LIN {X 0,Y 720.163,Z 331.517,A -85,B 0,C 180,E1 -1485.703,E2 -1485.703} C_VEL
LIN {X 0,Y 720.147,Z 331.521,A -85,B 0,C 180,E1 -1488.211,E2 -1488.211} C_VEL
LIN {X 0,Y 720.224,Z 331.521,A -85,B 0,C 180,E1 -1491.031,E2 -1491.031} C_VEL
LIN {X 0,Y 720.178,Z 331.657,A -85,B 0,C 180,E1 -1491.842,E2 -1491.842} C_VEL
LIN {X 0,Y 724.726,Z 343.937,A -85,B 0,C 180,E1 -1493.02,E2 -1493.02} C_VEL
LIN {X 0,Y 724.3,Z 377.381,A -85,B 0,C 180,E1 -1495.364,E2 -1495.364} C_VEL
LIN {X 0,Y 726.478,Z 386.978,A -85,B 0,C 180,E1 -1495.595,E2 -1495.595} C_VEL
LIN {X 0,Y 725.424,Z 646.257,A -85,B 0,C 180,E1 -1498.535,E2 -1498.535} C_VEL
LIN {X 0,Y 724.936,Z 767.062,A -85,B 0,C 180,E1 -1499.901,E2 -1499.901} C_VEL
LIN {X 0,Y 724.615,Z 792.765,A -85,B 0,C 180,E1 -1500.336,E2 -1500.336} C_VEL
LIN {X 0,Y 724.343,Z 814.335,A -85,B 0,C 180,E1 -1500.838,E2 -1500.838} C_VEL
LIN {X 0,Y 723.978,Z 838.569,A -85,B 0,C 180,E1 -1501.544,E2 -1501.544} C_VEL
LIN {X 0,Y 723.547,Z 860.48,A -85,B 0,C 180,E1 -1502.333,E2 -1502.333} C_VEL
LIN {X 0,Y 723.146,Z 883.178,A -85,B 0,C 180,E1 -1503.296,E2 -1503.296} C_VEL
LIN {X 0,Y 722.632,Z 904.751,A -85,B 0,C 180,E1 -1504.38,E2 -1504.38} C_VEL
LIN {X 0,Y 722.216,Z 925.848,A -85,B 0,C 180,E1 -1505.596,E2 -1505.596} C_VEL
LIN {X 0,Y 721.746,Z 945.563,A -85,B 0,C 180,E1 -1506.911,E2 -1506.911} C_VEL
LIN {X 0,Y 721.365,Z 964.777,A -85,B 0,C 180,E1 -1508.364,E2 -1508.364} C_VEL
LIN {X 0,Y 721.013,Z 981.39,A -85,B 0,C 180,E1 -1509.799,E2 -1509.799} C_VEL
LIN {X 0,Y 720.713,Z 998.517,A -85,B 0,C 180,E1 -1511.476,E2 -1511.476} C_VEL
LIN {X 0,Y 720.475,Z 1012.01,A -85,B 0,C 180,E1 -1512.982,E2 -1512.982} C_VEL
LIN {X 0,Y 720.287,Z 1026.218,A -85,B 0,C 180,E1 -1514.789,E2 -1514.789} C_VEL
LIN {X 0,Y 720.15,Z 1037.315,A -85,B 0,C 180,E1 -1516.429,E2 -1516.429} C_VEL
LIN {X 0,Y 720.044,Z 1047.962,A -85,B 0,C 180,E1 -1518.238,E2 -1518.238} C_VEL
LIN {X 0,Y 719.961,Z 1056.892,A -85,B 0,C 180,E1 -1520.083,E2 -1520.083} C_VEL
LIN {X 0,Y 719.941,Z 1063.423,A -85,B 0,C 180,E1 -1521.695,E2 -1521.695} C_VEL
LIN {X 0,Y 719.913,Z 1069.864,A -85,B 0,C 180,E1 -1523.701,E2 -1523.701} C_VEL
LIN {X 0,Y 719.916,Z 1073.813,A -85,B 0,C 180,E1 -1525.379,E2 -1525.379} C_VEL
LIN {X 0,Y 719.907,Z 1076.797,A -85,B 0,C 180,E1 -1527.214,E2 -1527.214} C_VEL
LIN {X 0,Y 719.9,Z 1078.284,A -85,B 0,C 180,E1 -1529.204,E2 -1529.204} C_VEL
LIN {X 0,Y 719.906,Z 1078.262,A -85,B 0,C 180,E1 -1530.875,E2 -1530.875} C_VEL
LIN {X 0,Y 719.913,Z 1076.572,A -85,B 0,C 180,E1 -1532.946,E2 -1532.946} C_VEL
LIN {X 0,Y 719.919,Z 1073.654,A -85,B 0,C 180,E1 -1534.7,E2 -1534.7} C_VEL
LIN {X 0,Y 719.908,Z 1069.015,A -85,B 0,C 180,E1 -1536.62,E2 -1536.62} C_VEL
LIN {X 0,Y 719.933,Z 1062.815,A -85,B 0,C 180,E1 -1538.466,E2 -1538.466} C_VEL
LIN {X 0,Y 719.974,Z 1056.182,A -85,B 0,C 180,E1 -1540.078,E2 -1540.078} C_VEL
LIN {X 0,Y 720.049,Z 1046.492,A -85,B 0,C 180,E1 -1542.022,E2 -1542.022} C_VEL
LIN {X 0,Y 720.154,Z 1036.797,A -85,B 0,C 180,E1 -1543.653,E2 -1543.653} C_VEL
LIN {X 0,Y 720.323,Z 1024.443,A -85,B 0,C 180,E1 -1545.457,E2 -1545.457} C_VEL
LIN {X 0,Y 720.483,Z 1011.221,A -85,B 0,C 180,E1 -1547.11,E2 -1547.11} C_VEL
LIN {X 0,Y 720.769,Z 996.177,A -85,B 0,C 180,E1 -1548.774,E2 -1548.774} C_VEL
LIN {X 0,Y 721.055,Z 979.534,A -85,B 0,C 180,E1 -1550.369,E2 -1550.369} C_VEL
LIN {X 0,Y 721.431,Z 961.606,A -85,B 0,C 180,E1 -1551.89,E2 -1551.89} C_VEL
LIN {X 0,Y 721.806,Z 943.238,A -85,B 0,C 180,E1 -1553.253,E2 -1553.253} C_VEL
LIN {X 0,Y 722.274,Z 921.437,A -85,B 0,C 180,E1 -1554.67,E2 -1554.67} C_VEL
LIN {X 0,Y 722.724,Z 901.529,A -85,B 0,C 180,E1 -1555.792,E2 -1555.792} C_VEL
LIN {X 0,Y 723.206,Z 878.258,A -85,B 0,C 180,E1 -1556.923,E2 -1556.923} C_VEL
LIN {X 0,Y 723.622,Z 857.112,A -85,B 0,C 180,E1 -1557.798,E2 -1557.798} C_VEL
LIN {X 0,Y 724.075,Z 832.967,A -85,B 0,C 180,E1 -1558.632,E2 -1558.632} C_VEL
LIN {X 0,Y 724.365,Z 811.106,A -85,B 0,C 180,E1 -1559.246,E2 -1559.246} C_VEL
LIN {X 0,Y 724.75,Z 786.453,A -85,B 0,C 180,E1 -1559.787,E2 -1559.787} C_VEL
LIN {X 0,Y 724.95,Z 763.825,A -85,B 0,C 180,E1 -1560.142,E2 -1560.142} C_VEL
LIN {X 0,Y 725.946,Z 508.893,A -85,B 0,C 180,E1 -1563.013,E2 -1563.013} C_VEL
LIN {X 0,Y 726.28,Z 385.255,A -85,B 0,C 180,E1 -1564.436,E2 -1564.436} C_VEL
LIN {X 0,Y 724.228,Z 376.686,A -85,B 0,C 180,E1 -1564.668,E2 -1564.668} C_VEL
LIN {X 0,Y 724.705,Z 343.754,A -85,B 0,C 180,E1 -1566.995,E2 -1566.995} C_VEL
LIN {X 0,Y 720.161,Z 331.519,A -85,B 0,C 180,E1 -1568.182,E2 -1568.182} C_VEL
LIN {X 0,Y 720.198,Z 331.523,A -85,B 0,C 180,E1 -1571.193,E2 -1571.193} C_VEL
LIN {X 0,Y 720.148,Z 331.519,A -85,B 0,C 180,E1 -1573.895,E2 -1573.895} C_VEL
LIN {X 0,Y 720.193,Z 331.516,A -85,B 0,C 180,E1 -1576.588,E2 -1576.588} C_VEL
LIN {X 0,Y 720.169,Z 331.519,A -85,B 0,C 180,E1 -1579.58,E2 -1579.58} C_VEL
LIN {X 0,Y 720.148,Z 331.518,A -85,B 0,C 180,E1 -1582.143,E2 -1582.143} C_VEL
LIN {X 0,Y 720.215,Z 331.502,A -85,B 0,C 180,E1 -1584.917,E2 -1584.917} C_VEL
LIN {X 0,Y 720.156,Z 331.518,A -85,B 0,C 180,E1 -1587.881,E2 -1587.881} C_VEL
LIN {X 0,Y 720.152,Z 331.517,A -85,B 0,C 180,E1 -1590.377,E2 -1590.377} C_VEL
LIN {X 0,Y 720.225,Z 331.513,A -85,B 0,C 180,E1 -1593.212,E2 -1593.212} C_VEL
LIN {X 0,Y 720.155,Z 331.517,A -85,B 0,C 180,E1 -1596.082,E2 -1596.082} C_VEL
LIN {X 0,Y 720.162,Z 331.516,A -85,B 0,C 180,E1 -1598.668,E2 -1598.668} C_VEL
LIN {X 0,Y 720.211,Z 331.523,A -85,B 0,C 180,E1 -1601.63,E2 -1601.63} C_VEL
LIN {X 0,Y 720.149,Z 331.517,A -85,B 0,C 180,E1 -1604.374,E2 -1604.374} C_VEL
LIN {X 0,Y 720.181,Z 331.515,A -85,B 0,C 180,E1 -1607.002,E2 -1607.002} C_VEL
LIN {X 0,Y 720.172,Z 331.521,A -85,B 0,C 180,E1 -1610.086,E2 -1610.086} C_VEL
LIN {X 0,Y 720.151,Z 331.513,A -85,B 0,C 180,E1 -1612.661,E2 -1612.661} C_VEL
LIN {X 0,Y 720.219,Z 331.515,A -85,B 0,C 180,E1 -1615.461,E2 -1615.461} C_VEL
LIN {X 0,Y 720.159,Z 331.519,A -85,B 0,C 180,E1 -1618.409,E2 -1618.409} C_VEL
LIN {X 0,Y 720.157,Z 331.516,A -85,B 0,C 180,E1 -1620.955,E2 -1620.955} C_VEL
LIN {X 0,Y 720.222,Z 331.517,A -85,B 0,C 180,E1 -1623.821,E2 -1623.821} C_VEL
LIN {X 0,Y 720.156,Z 331.515,A -85,B 0,C 180,E1 -1626.618,E2 -1626.618} C_VEL
LIN {X 0,Y 720.164,Z 331.516,A -85,B 0,C 180,E1 -1629.19,E2 -1629.19} C_VEL
LIN {X 0,Y 720.209,Z 331.521,A -85,B 0,C 180,E1 -1632.208,E2 -1632.208} C_VEL
LIN {X 0,Y 720.153,Z 331.516,A -85,B 0,C 180,E1 -1634.966,E2 -1634.966} C_VEL
LIN {X 0,Y 720.21,Z 331.52,A -85,B 0,C 180,E1 -1636.267,E2 -1636.267} C_VEL
LIN {X 0,Y 719.173,Z 331.652,A -85,B 0,C 180,E1 -1636.88,E2 -1636.88} C_VEL
LIN {X 0,Y 712.742,Z 332.446,A -85,B 0,C 180,E1 -1638.597,E2 -1638.597} C_VEL
LIN {X 0,Y 712.215,Z 332.505,A -85,B 0,C 180,E1 -1639.043,E2 -1639.043} C_VEL
LIN {X 0,Y 712.276,Z 332.502,A -85,B 0,C 180,E1 -1641.84,E2 -1641.84} C_VEL
LIN {X 0,Y 712.226,Z 332.509,A -85,B 0,C 180,E1 -1644.82,E2 -1644.82} C_VEL
LIN {X 0,Y 712.226,Z 332.503,A -85,B 0,C 180,E1 -1647.469,E2 -1647.469} C_VEL
LIN {X 0,Y 712.279,Z 332.508,A -85,B 0,C 180,E1 -1650.467,E2 -1650.467} C_VEL
LIN {X 0,Y 712.217,Z 332.507,A -85,B 0,C 180,E1 -1653.294,E2 -1653.294} C_VEL
LIN {X 0,Y 712.28,Z 332.503,A -85,B 0,C 180,E1 -1656.128,E2 -1656.128} C_VEL
LIN {X 0,Y 712.227,Z 332.509,A -85,B 0,C 180,E1 -1659.076,E2 -1659.076} C_VEL
LIN {X 0,Y 712.227,Z 332.506,A -85,B 0,C 180,E1 -1661.717,E2 -1661.717} C_VEL
LIN {X 0,Y 712.274,Z 332.509,A -85,B 0,C 180,E1 -1664.739,E2 -1664.739} C_VEL
LIN {X 0,Y 712.218,Z 332.509,A -85,B 0,C 180,E1 -1667.524,E2 -1667.524} C_VEL
LIN {X 0,Y 712.278,Z 332.506,A -85,B 0,C 180,E1 -1670.303,E2 -1670.303} C_VEL
LIN {X 0,Y 712.232,Z 332.508,A -85,B 0,C 180,E1 -1673.285,E2 -1673.285} C_VEL
LIN {X 0,Y 712.237,Z 332.645,A -85,B 0,C 180,E1 -1673.57,E2 -1673.57} C_VEL
LIN {X 0,Y 716.875,Z 346.54,A -85,B 0,C 180,E1 -1674.925,E2 -1674.925} C_VEL
LIN {X 0,Y 717.007,Z 348.113,A -85,B 0,C 180,E1 -1675.014,E2 -1675.014} C_VEL
LIN {X 0,Y 719.82,Z 359.371,A -85,B 0,C 180,E1 -1675.305,E2 -1675.305} C_VEL
LIN {X 0,Y 718.682,Z 598.601,A -85,B 0,C 180,E1 -1678.047,E2 -1678.047} C_VEL
LIN {X 0,Y 718.006,Z 736.954,A -85,B 0,C 180,E1 -1679.623,E2 -1679.623} C_VEL
LIN {X 0,Y 717.638,Z 762.534,A -85,B 0,C 180,E1 -1680.059,E2 -1680.059} C_VEL
LIN {X 0,Y 717.293,Z 784.195,A -85,B 0,C 180,E1 -1680.564,E2 -1680.564} C_VEL
LIN {X 0,Y 716.857,Z 808.586,A -85,B 0,C 180,E1 -1681.281,E2 -1681.281} C_VEL
LIN {X 0,Y 716.344,Z 830.47,A -85,B 0,C 180,E1 -1682.075,E2 -1682.075} C_VEL
LIN {X 0,Y 715.848,Z 853.086,A -85,B 0,C 180,E1 -1683.043,E2 -1683.043} C_VEL
LIN {X 0,Y 715.244,Z 874.745,A -85,B 0,C 180,E1 -1684.141,E2 -1684.141} C_VEL
LIN {X 0,Y 714.721,Z 895.739,A -85,B 0,C 180,E1 -1685.361,E2 -1685.361} C_VEL
LIN {X 0,Y 714.171,Z 915.623,A -85,B 0,C 180,E1 -1686.701,E2 -1686.701} C_VEL
LIN {X 0,Y 713.69,Z 934.764,A -85,B 0,C 180,E1 -1688.163,E2 -1688.163} C_VEL
LIN {X 0,Y 713.286,Z 950.904,A -85,B 0,C 180,E1 -1689.571,E2 -1689.571} C_VEL
LIN {X 0,Y 712.928,Z 967.586,A -85,B 0,C 180,E1 -1691.209,E2 -1691.209} C_VEL
LIN {X 0,Y 712.6,Z 982.184,A -85,B 0,C 180,E1 -1692.854,E2 -1692.854} C_VEL
LIN {X 0,Y 712.364,Z 996.488,A -85,B 0,C 180,E1 -1694.7,E2 -1694.7} C_VEL
LIN {X 0,Y 712.199,Z 1007.556,A -85,B 0,C 180,E1 -1696.358,E2 -1696.358} C_VEL
LIN {X 0,Y 712.08,Z 1018.068,A -85,B 0,C 180,E1 -1698.17,E2 -1698.17} C_VEL
LIN {X 0,Y 711.984,Z 1026.697,A -85,B 0,C 180,E1 -1699.971,E2 -1699.971} C_VEL
LIN {X 0,Y 711.943,Z 1033.255,A -85,B 0,C 180,E1 -1701.601,E2 -1701.601} C_VEL
LIN {X 0,Y 711.921,Z 1039.75,A -85,B 0,C 180,E1 -1703.63,E2 -1703.63} C_VEL
LIN {X 0,Y 711.915,Z 1043.884,A -85,B 0,C 180,E1 -1705.408,E2 -1705.408} C_VEL
LIN {X 0,Y 711.896,Z 1046.847,A -85,B 0,C 180,E1 -1707.263,E2 -1707.263} C_VEL
LIN {X 0,Y 711.901,Z 1048.272,A -85,B 0,C 180,E1 -1709.195,E2 -1709.195} C_VEL
LIN {X 0,Y 711.906,Z 1048.274,A -85,B 0,C 180,E1 -1710.885,E2 -1710.885} C_VEL
LIN {X 0,Y 711.905,Z 1046.747,A -85,B 0,C 180,E1 -1712.898,E2 -1712.898} C_VEL
LIN {X 0,Y 711.915,Z 1043.902,A -85,B 0,C 180,E1 -1714.673,E2 -1714.673} C_VEL
LIN {X 0,Y 711.914,Z 1039.772,A -85,B 0,C 180,E1 -1716.451,E2 -1716.451} C_VEL
LIN {X 0,Y 711.94,Z 1033.287,A -85,B 0,C 180,E1 -1718.48,E2 -1718.48} C_VEL
LIN {X 0,Y 711.991,Z 1026.718,A -85,B 0,C 180,E1 -1720.114,E2 -1720.114} C_VEL
LIN {X 0,Y 712.085,Z 1017.658,A -85,B 0,C 180,E1 -1721.995,E2 -1721.995} C_VEL
LIN {X 0,Y 712.204,Z 1007.079,A -85,B 0,C 180,E1 -1723.808,E2 -1723.808} C_VEL
LIN {X 0,Y 712.406,Z 994.78,A -85,B 0,C 180,E1 -1725.633,E2 -1725.633} C_VEL
LIN {X 0,Y 712.628,Z 980.892,A -85,B 0,C 180,E1 -1727.389,E2 -1727.389} C_VEL
LIN {X 0,Y 712.956,Z 965.781,A -85,B 0,C 180,E1 -1729.073,E2 -1729.073} C_VEL
LIN {X 0,Y 713.31,Z 950.02,A -85,B 0,C 180,E1 -1730.6,E2 -1730.6} C_VEL
LIN {X 0,Y 713.758,Z 932.179,A -85,B 0,C 180,E1 -1732.138,E2 -1732.138} C_VEL
LIN {X 0,Y 714.223,Z 913.86,A -85,B 0,C 180,E1 -1733.515,E2 -1733.515} C_VEL
LIN {X 0,Y 714.759,Z 893.636,A -85,B 0,C 180,E1 -1734.858,E2 -1734.858} C_VEL
LIN {X 0,Y 715.297,Z 873.155,A -85,B 0,C 180,E1 -1736.036,E2 -1736.036} C_VEL
LIN {X 0,Y 715.891,Z 850.245,A -85,B 0,C 180,E1 -1737.176,E2 -1737.176} C_VEL
LIN {X 0,Y 716.368,Z 829.357,A -85,B 0,C 180,E1 -1738.059,E2 -1738.059} C_VEL
LIN {X 0,Y 716.936,Z 805.882,A -85,B 0,C 180,E1 -1738.898,E2 -1738.898} C_VEL
LIN {X 0,Y 717.311,Z 782.472,A -85,B 0,C 180,E1 -1739.571,E2 -1739.571} C_VEL
LIN {X 0,Y 717.764,Z 758.503,A -85,B 0,C 180,E1 -1740.115,E2 -1740.115} C_VEL
LIN {X 0,Y 718.018,Z 734.505,A -85,B 0,C 180,E1 -1740.499,E2 -1740.499} C_VEL
LIN {X 0,Y 719.269,Z 474.983,A -85,B 0,C 180,E1 -1743.45,E2 -1743.45} C_VEL
LIN {X 0,Y 719.631,Z 357.815,A -85,B 0,C 180,E1 -1744.814,E2 -1744.814} C_VEL
LIN {X 0,Y 716.852,Z 347.387,A -85,B 0,C 180,E1 -1745.101,E2 -1745.101} C_VEL
LIN {X 0,Y 716.411,Z 344.69,A -85,B 0,C 180,E1 -1745.335,E2 -1745.335} C_VEL
LIN {X 0,Y 712.213,Z 332.514,A -85,B 0,C 180,E1 -1746.555,E2 -1746.555} C_VEL
LIN {X 0,Y 712.284,Z 332.507,A -85,B 0,C 180,E1 -1749.384,E2 -1749.384} C_VEL
LIN {X 0,Y 712.216,Z 332.509,A -85,B 0,C 180,E1 -1752.28,E2 -1752.28} C_VEL
LIN {X 0,Y 712.218,Z 332.502,A -85,B 0,C 180,E1 -1754.848,E2 -1754.848} C_VEL
LIN {X 0,Y 712.272,Z 332.494,A -85,B 0,C 180,E1 -1757.834,E2 -1757.834} C_VEL
LIN {X 0,Y 712.21,Z 332.507,A -85,B 0,C 180,E1 -1760.611,E2 -1760.611} C_VEL
LIN {X 0,Y 712.248,Z 332.508,A -85,B 0,C 180,E1 -1763.283,E2 -1763.283} C_VEL
LIN {X 0,Y 712.227,Z 332.505,A -85,B 0,C 180,E1 -1766.357,E2 -1766.357} C_VEL
LIN {X 0,Y 712.215,Z 332.506,A -85,B 0,C 180,E1 -1768.986,E2 -1768.986} C_VEL
LIN {X 0,Y 712.284,Z 332.503,A -85,B 0,C 180,E1 -1771.857,E2 -1771.857} C_VEL
LIN {X 0,Y 712.213,Z 332.507,A -85,B 0,C 180,E1 -1774.706,E2 -1774.706} C_VEL
LIN {X 0,Y 712.223,Z 332.507,A -85,B 0,C 180,E1 -1777.29,E2 -1777.29} C_VEL
LIN {X 0,Y 712.261,Z 332.501,A -85,B 0,C 180,E1 -1780.311,E2 -1780.311} C_VEL
LIN {X 0,Y 712.209,Z 332.507,A -85,B 0,C 180,E1 -1783.021,E2 -1783.021} C_VEL
LIN {X 0,Y 712.251,Z 332.507,A -85,B 0,C 180,E1 -1785.695,E2 -1785.695} C_VEL
LIN {X 0,Y 712.225,Z 332.501,A -85,B 0,C 180,E1 -1788.747,E2 -1788.747} C_VEL
LIN {X 0,Y 712.213,Z 332.508,A -85,B 0,C 180,E1 -1791.36,E2 -1791.36} C_VEL
LIN {X 0,Y 712.285,Z 332.506,A -85,B 0,C 180,E1 -1794.199,E2 -1794.199} C_VEL
LIN {X 0,Y 712.212,Z 332.506,A -85,B 0,C 180,E1 -1797.103,E2 -1797.103} C_VEL
LIN {X 0,Y 712.224,Z 332.506,A -85,B 0,C 180,E1 -1799.678,E2 -1799.678} C_VEL
LIN {X 0,Y 712.252,Z 332.499,A -85,B 0,C 180,E1 -1802.736,E2 -1802.736} C_VEL
LIN {X 0,Y 712.209,Z 332.508,A -85,B 0,C 180,E1 -1805.397,E2 -1805.397} C_VEL
LIN {X 0,Y 712.25,Z 332.507,A -85,B 0,C 180,E1 -1808.07,E2 -1808.07} C_VEL
LIN {X 0,Y 712.228,Z 332.504,A -85,B 0,C 180,E1 -1811.092,E2 -1811.092} C_VEL
LIN {X 0,Y 712.211,Z 332.507,A -85,B 0,C 180,E1 -1813.708,E2 -1813.708} C_VEL
LIN {X 0,Y 712.284,Z 332.504,A -85,B 0,C 180,E1 -1816.557,E2 -1816.557} C_VEL
LIN {X 0,Y 712.212,Z 332.506,A -85,B 0,C 180,E1 -1819.435,E2 -1819.435} C_VEL
LIN {X 0,Y 712.22,Z 332.507,A -85,B 0,C 180,E1 -1822.015,E2 -1822.015} C_VEL
LIN {X 0,Y 712.269,Z 332.503,A -85,B 0,C 180,E1 -1824.996,E2 -1824.996} C_VEL
LIN {X 0,Y 712.209,Z 332.505,A -85,B 0,C 180,E1 -1827.691,E2 -1827.691} C_VEL
LIN {X 0,Y 712.234,Z 332.511,A -85,B 0,C 180,E1 -1830.301,E2 -1830.301} C_VEL
LIN {X 0,Y 712.235,Z 332.505,A -85,B 0,C 180,E1 -1833.389,E2 -1833.389} C_VEL
LIN {X 0,Y 712.209,Z 332.509,A -85,B 0,C 180,E1 -1835.933,E2 -1835.933} C_VEL
LIN {X 0,Y 712.266,Z 332.512,A -85,B 0,C 180,E1 -1838.692,E2 -1838.692} C_VEL
LIN {X 0,Y 712.221,Z 332.504,A -85,B 0,C 180,E1 -1841.679,E2 -1841.679} C_VEL
LIN {X 0,Y 712.213,Z 332.508,A -85,B 0,C 180,E1 -1844.275,E2 -1844.275} C_VEL
LIN {X 0,Y 712.28,Z 332.506,A -85,B 0,C 180,E1 -1847.201,E2 -1847.201} C_VEL
LIN {X 0,Y 712.211,Z 332.512,A -85,B 0,C 180,E1 -1849.984,E2 -1849.984} C_VEL
LIN {X 0,Y 712.303,Z 332.751,A -85,B 0,C 180,E1 -1851.434,E2 -1851.434} C_VEL
LIN {X 0,Y 717.694,Z 347.21,A -85,B 0,C 180,E1 -1852.836,E2 -1852.836} C_VEL
LIN {X 0,Y 717.276,Z 377.476,A -85,B 0,C 180,E1 -1854.976,E2 -1854.976} C_VEL
LIN {X 0,Y 719.862,Z 388.764,A -85,B 0,C 180,E1 -1855.255,E2 -1855.255} C_VEL
LIN {X 0,Y 718.587,Z 648.03,A -85,B 0,C 180,E1 -1858.222,E2 -1858.222} C_VEL
LIN {X 0,Y 718.004,Z 767.169,A -85,B 0,C 180,E1 -1859.581,E2 -1859.581} C_VEL
LIN {X 0,Y 717.629,Z 792.892,A -85,B 0,C 180,E1 -1860.021,E2 -1860.021} C_VEL
LIN {X 0,Y 717.29,Z 814.457,A -85,B 0,C 180,E1 -1860.526,E2 -1860.526} C_VEL
LIN {X 0,Y 716.861,Z 838.566,A -85,B 0,C 180,E1 -1861.235,E2 -1861.235} C_VEL
LIN {X 0,Y 716.339,Z 860.484,A -85,B 0,C 180,E1 -1862.031,E2 -1862.031} C_VEL
LIN {X 0,Y 715.831,Z 883.581,A -85,B 0,C 180,E1 -1863.022,E2 -1863.022} C_VEL
LIN {X 0,Y 715.246,Z 904.755,A -85,B 0,C 180,E1 -1864.096,E2 -1864.096} C_VEL
LIN {X 0,Y 714.719,Z 925.754,A -85,B 0,C 180,E1 -1865.317,E2 -1865.317} C_VEL
LIN {X 0,Y 714.178,Z 945.151,A -85,B 0,C 180,E1 -1866.622,E2 -1866.622} C_VEL
LIN {X 0,Y 713.724,Z 963.808,A -85,B 0,C 180,E1 -1868.038,E2 -1868.038} C_VEL
LIN {X 0,Y 713.296,Z 980.461,A -85,B 0,C 180,E1 -1869.485,E2 -1869.485} C_VEL
LIN {X 0,Y 712.939,Z 996.965,A -85,B 0,C 180,E1 -1871.096,E2 -1871.096} C_VEL
LIN {X 0,Y 712.623,Z 1011.222,A -85,B 0,C 180,E1 -1872.695,E2 -1872.695} C_VEL
LIN {X 0,Y 712.408,Z 1025.06,A -85,B 0,C 180,E1 -1874.45,E2 -1874.45} C_VEL
LIN {X 0,Y 712.209,Z 1036.796,A -85,B 0,C 180,E1 -1876.192,E2 -1876.192} C_VEL
LIN {X 0,Y 712.082,Z 1046.948,A -85,B 0,C 180,E1 -1877.923,E2 -1877.923} C_VEL
LIN {X 0,Y 711.99,Z 1056.524,A -85,B 0,C 180,E1 -1879.886,E2 -1879.886} C_VEL
LIN {X 0,Y 711.94,Z 1063.119,A -85,B 0,C 180,E1 -1881.52,E2 -1881.52} C_VEL
LIN {X 0,Y 711.909,Z 1069.451,A -85,B 0,C 180,E1 -1883.467,E2 -1883.467} C_VEL
LIN {X 0,Y 711.918,Z 1073.813,A -85,B 0,C 180,E1 -1885.327,E2 -1885.327} C_VEL
LIN {X 0,Y 711.908,Z 1076.797,A -85,B 0,C 180,E1 -1887.182,E2 -1887.182} C_VEL
LIN {X 0,Y 711.901,Z 1078.284,A -85,B 0,C 180,E1 -1889.195,E2 -1889.195} C_VEL
LIN {X 0,Y 711.906,Z 1078.262,A -85,B 0,C 180,E1 -1890.885,E2 -1890.885} C_VEL
LIN {X 0,Y 711.913,Z 1076.572,A -85,B 0,C 180,E1 -1892.979,E2 -1892.979} C_VEL
LIN {X 0,Y 711.919,Z 1073.655,A -85,B 0,C 180,E1 -1894.753,E2 -1894.753} C_VEL
LIN {X 0,Y 711.913,Z 1069.015,A -85,B 0,C 180,E1 -1896.694,E2 -1896.694} C_VEL
LIN {X 0,Y 711.938,Z 1062.815,A -85,B 0,C 180,E1 -1898.562,E2 -1898.562} C_VEL
LIN {X 0,Y 712.001,Z 1056.183,A -85,B 0,C 180,E1 -1900.192,E2 -1900.192} C_VEL
LIN {X 0,Y 712.095,Z 1046.032,A -85,B 0,C 180,E1 -1902.241,E2 -1902.241} C_VEL
LIN {X 0,Y 712.214,Z 1036.279,A -85,B 0,C 180,E1 -1903.891,E2 -1903.891} C_VEL
LIN {X 0,Y 712.423,Z 1023.807,A -85,B 0,C 180,E1 -1905.716,E2 -1905.716} C_VEL
LIN {X 0,Y 712.64,Z 1010.515,A -85,B 0,C 180,E1 -1907.389,E2 -1907.389} C_VEL
LIN {X 0,Y 712.961,Z 995.334,A -85,B 0,C 180,E1 -1909.073,E2 -1909.073} C_VEL
LIN {X 0,Y 713.319,Z 979.534,A -85,B 0,C 180,E1 -1910.6,E2 -1910.6} C_VEL
LIN {X 0,Y 713.766,Z 961.607,A -85,B 0,C 180,E1 -1912.138,E2 -1912.138} C_VEL
LIN {X 0,Y 714.239,Z 943.238,A -85,B 0,C 180,E1 -1913.514,E2 -1913.514} C_VEL
LIN {X 0,Y 714.782,Z 922.167,A -85,B 0,C 180,E1 -1914.901,E2 -1914.901} C_VEL
LIN {X 0,Y 715.321,Z 902.335,A -85,B 0,C 180,E1 -1916.035,E2 -1916.035} C_VEL
LIN {X 0,Y 715.904,Z 879.256,A -85,B 0,C 180,E1 -1917.175,E2 -1917.175} C_VEL
LIN {X 0,Y 716.401,Z 858.24,A -85,B 0,C 180,E1 -1918.057,E2 -1918.057} C_VEL
LIN {X 0,Y 716.951,Z 834.44,A -85,B 0,C 180,E1 -1918.897,E2 -1918.897} C_VEL
LIN {X 0,Y 717.314,Z 811.862,A -85,B 0,C 180,E1 -1919.542,E2 -1919.542} C_VEL
LIN {X 0,Y 717.775,Z 787.54,A -85,B 0,C 180,E1 -1920.087,E2 -1920.087} C_VEL
LIN {X 0,Y 718.02,Z 764.119,A -85,B 0,C 180,E1 -1920.459,E2 -1920.459} C_VEL
LIN {X 0,Y 719.22,Z 511.246,A -85,B 0,C 180,E1 -1923.334,E2 -1923.334} C_VEL
LIN {X 0,Y 719.678,Z 387.122,A -85,B 0,C 180,E1 -1924.775,E2 -1924.775} C_VEL
LIN {X 0,Y 717.183,Z 376.686,A -85,B 0,C 180,E1 -1925.058,E2 -1925.058} C_VEL
LIN {X 0,Y 717.694,Z 347.21,A -85,B 0,C 180,E1 -1927.164,E2 -1927.164} C_VEL
LIN {X 0,Y 712.275,Z 332.499,A -85,B 0,C 180,E1 -1928.608,E2 -1928.608} C_VEL
LIN {X 0,Y 712.219,Z 332.511,A -85,B 0,C 180,E1 -1931.558,E2 -1931.558} C_VEL
LIN {X 0,Y 712.213,Z 332.508,A -85,B 0,C 180,E1 -1934.134,E2 -1934.134} C_VEL
LIN {X 0,Y 712.282,Z 332.509,A -85,B 0,C 180,E1 -1937.001,E2 -1937.001} C_VEL
LIN {X 0,Y 712.215,Z 332.507,A -85,B 0,C 180,E1 -1939.794,E2 -1939.794} C_VEL
LIN {X 0,Y 712.22,Z 332.506,A -85,B 0,C 180,E1 -1942.36,E2 -1942.36} C_VEL
LIN {X 0,Y 712.269,Z 332.499,A -85,B 0,C 180,E1 -1945.351,E2 -1945.351} C_VEL
LIN {X 0,Y 712.21,Z 332.506,A -85,B 0,C 180,E1 -1948.043,E2 -1948.043} C_VEL
LIN {X 0,Y 712.236,Z 332.504,A -85,B 0,C 180,E1 -1950.669,E2 -1950.669} C_VEL
LIN {X 0,Y 712.236,Z 332.51,A -85,B 0,C 180,E1 -1953.776,E2 -1953.776} C_VEL
LIN {X 0,Y 712.213,Z 332.504,A -85,B 0,C 180,E1 -1956.414,E2 -1956.414} C_VEL
LIN {X 0,Y 712.281,Z 332.504,A -85,B 0,C 180,E1 -1959.215,E2 -1959.215} C_VEL
LIN {X 0,Y 712.219,Z 332.508,A -85,B 0,C 180,E1 -1962.147,E2 -1962.147} C_VEL
LIN {X 0,Y 712.219,Z 332.504,A -85,B 0,C 180,E1 -1964.696,E2 -1964.696} C_VEL
LIN {X 0,Y 712.282,Z 332.507,A -85,B 0,C 180,E1 -1967.597,E2 -1967.597} C_VEL
LIN {X 0,Y 712.214,Z 332.508,A -85,B 0,C 180,E1 -1970.383,E2 -1970.383} C_VEL
LIN {X 0,Y 712.231,Z 332.499,A -85,B 0,C 180,E1 -1972.999,E2 -1972.999} C_VEL
LIN {X 0,Y 712.25,Z 332.507,A -85,B 0,C 180,E1 -1976.056,E2 -1976.056} C_VEL
LIN {X 0,Y 712.214,Z 332.506,A -85,B 0,C 180,E1 -1978.713,E2 -1978.713} C_VEL
LIN {X 0,Y 712.272,Z 332.502,A -85,B 0,C 180,E1 -1981.448,E2 -1981.448} C_VEL
LIN {X 0,Y 712.228,Z 332.509,A -85,B 0,C 180,E1 -1984.428,E2 -1984.428} C_VEL
LIN {X 0,Y 712.217,Z 332.501,A -85,B 0,C 180,E1 -1987.016,E2 -1987.016} C_VEL
LIN {X 0,Y 712.283,Z 332.506,A -85,B 0,C 180,E1 -1989.861,E2 -1989.861} C_VEL
LIN {X 0,Y 712.22,Z 332.508,A -85,B 0,C 180,E1 -1992.733,E2 -1992.733} C_VEL
LIN {X 0,Y 712.228,Z 332.503,A -85,B 0,C 180,E1 -1995.319,E2 -1995.319} C_VEL
LIN {X 0,Y 712.267,Z 332.51,A -85,B 0,C 180,E1 -1998.328,E2 -1998.328} C_VEL
LIN {X 0,Y 712.215,Z 332.505,A -85,B 0,C 180,E1 -1999.043,E2 -1999.043} C_VEL
LIN {X 0,Y 711.23,Z 332.631,A -85,B 0,C 180,E1 -1999.663,E2 -1999.663} C_VEL
LIN {X 0,Y 704.844,Z 333.426,A -85,B 0,C 180,E1 -2001.399,E2 -2001.399} C_VEL
LIN {X 0,Y 704.338,Z 333.491,A -85,B 0,C 180,E1 -2001.85,E2 -2001.85} C_VEL
LIN {X 0,Y 704.285,Z 333.497,A -85,B 0,C 180,E1 -2004.85,E2 -2004.85} C_VEL
LIN {X 0,Y 704.288,Z 333.492,A -85,B 0,C 180,E1 -2007.478,E2 -2007.478} C_VEL
LIN {X 0,Y 704.336,Z 333.496,A -85,B 0,C 180,E1 -2010.491,E2 -2010.491} C_VEL
LIN {X 0,Y 704.279,Z 333.496,A -85,B 0,C 180,E1 -2013.329,E2 -2013.329} C_VEL
LIN {X 0,Y 704.344,Z 333.493,A -85,B 0,C 180,E1 -2016.197,E2 -2016.197} C_VEL
LIN {X 0,Y 704.288,Z 333.498,A -85,B 0,C 180,E1 -2019.077,E2 -2019.077} C_VEL
LIN {X 0,Y 704.291,Z 333.495,A -85,B 0,C 180,E1 -2021.747,E2 -2021.747} C_VEL
LIN {X 0,Y 704.33,Z 333.497,A -85,B 0,C 180,E1 -2024.78,E2 -2024.78} C_VEL
LIN {X 0,Y 704.279,Z 333.499,A -85,B 0,C 180,E1 -2027.484,E2 -2027.484} C_VEL
LIN {X 0,Y 704.339,Z 333.495,A -85,B 0,C 180,E1 -2030.296,E2 -2030.296} C_VEL
LIN {X 0,Y 704.32,Z 333.634,A -85,B 0,C 180,E1 -2033.172,E2 -2033.172} C_VEL
LIN {X 0,Y 709.368,Z 347.884,A -85,B 0,C 180,E1 -2034.578,E2 -2034.578} C_VEL
LIN {X 0,Y 711.003,Z 352.12,A -85,B 0,C 180,E1 -2034.723,E2 -2034.723} C_VEL
LIN {X 0,Y 713.229,Z 361.085,A -85,B 0,C 180,E1 -2034.958,E2 -2034.958} C_VEL
LIN {X 0,Y 711.884,Z 600.56,A -85,B 0,C 180,E1 -2037.728,E2 -2037.728} C_VEL
LIN {X 0,Y 711.097,Z 737.105,A -85,B 0,C 180,E1 -2039.298,E2 -2039.298} C_VEL
LIN {X 0,Y 710.679,Z 762.714,A -85,B 0,C 180,E1 -2039.738,E2 -2039.738} C_VEL
LIN {X 0,Y 710.263,Z 784.404,A -85,B 0,C 180,E1 -2040.249,E2 -2040.249} C_VEL
LIN {X 0,Y 709.759,Z 808.599,A -85,B 0,C 180,E1 -2040.966,E2 -2040.966} C_VEL
LIN {X 0,Y 709.163,Z 830.517,A -85,B 0,C 180,E1 -2041.768,E2 -2041.768} C_VEL
LIN {X 0,Y 708.557,Z 853.296,A -85,B 0,C 180,E1 -2042.753,E2 -2042.753} C_VEL
LIN {X 0,Y 707.875,Z 874.758,A -85,B 0,C 180,E1 -2043.851,E2 -2043.851} C_VEL
LIN {X 0,Y 707.237,Z 895.744,A -85,B 0,C 180,E1 -2045.083,E2 -2045.083} C_VEL
LIN {X 0,Y 706.626,Z 915.042,A -85,B 0,C 180,E1 -2046.394,E2 -2046.394} C_VEL
LIN {X 0,Y 706.047,Z 934.257,A -85,B 0,C 180,E1 -2047.87,E2 -2047.87} C_VEL
LIN {X 0,Y 705.56,Z 950.911,A -85,B 0,C 180,E1 -2049.337,E2 -2049.337} C_VEL
LIN {X 0,Y 705.123,Z 967.338,A -85,B 0,C 180,E1 -2050.965,E2 -2050.965} C_VEL
LIN {X 0,Y 704.759,Z 981.558,A -85,B 0,C 180,E1 -2052.581,E2 -2052.581} C_VEL
LIN {X 0,Y 704.49,Z 995.336,A -85,B 0,C 180,E1 -2054.356,E2 -2054.356} C_VEL
LIN {X 0,Y 704.268,Z 1007.041,A -85,B 0,C 180,E1 -2056.117,E2 -2056.117} C_VEL
LIN {X 0,Y 704.117,Z 1017.618,A -85,B 0,C 180,E1 -2057.951,E2 -2057.951} C_VEL
LIN {X 0,Y 704.01,Z 1026.7,A -85,B 0,C 180,E1 -2059.857,E2 -2059.857} C_VEL
LIN {X 0,Y 703.948,Z 1033.257,A -85,B 0,C 180,E1 -2061.505,E2 -2061.505} C_VEL
LIN {X 0,Y 703.922,Z 1039.544,A -85,B 0,C 180,E1 -2063.475,E2 -2063.475} C_VEL
LIN {X 0,Y 703.909,Z 1043.726,A -85,B 0,C 180,E1 -2065.274,E2 -2065.274} C_VEL
LIN {X 0,Y 703.911,Z 1046.51,A -85,B 0,C 180,E1 -2066.987,E2 -2066.987} C_VEL
LIN {X 0,Y 703.907,Z 1048.25,A -85,B 0,C 180,E1 -2069.105,E2 -2069.105} C_VEL
LIN {X 0,Y 703.902,Z 1048.296,A -85,B 0,C 180,E1 -2070.814,E2 -2070.814} C_VEL
LIN {X 0,Y 703.898,Z 1046.972,A -85,B 0,C 180,E1 -2072.768,E2 -2072.768} C_VEL
LIN {X 0,Y 703.916,Z 1044.06,A -85,B 0,C 180,E1 -2074.644,E2 -2074.644} C_VEL
LIN {X 0,Y 703.918,Z 1040.184,A -85,B 0,C 180,E1 -2076.361,E2 -2076.361} C_VEL
LIN {X 0,Y 703.95,Z 1033.892,A -85,B 0,C 180,E1 -2078.413,E2 -2078.413} C_VEL
LIN {X 0,Y 704.006,Z 1027.087,A -85,B 0,C 180,E1 -2080.144,E2 -2080.144} C_VEL
LIN {X 0,Y 704.115,Z 1018.105,A -85,B 0,C 180,E1 -2082.049,E2 -2082.049} C_VEL
LIN {X 0,Y 704.259,Z 1007.596,A -85,B 0,C 180,E1 -2083.883,E2 -2083.883} C_VEL
LIN {X 0,Y 704.475,Z 995.95,A -85,B 0,C 180,E1 -2085.645,E2 -2085.645} C_VEL
LIN {X 0,Y 704.741,Z 982.305,A -85,B 0,C 180,E1 -2087.42,E2 -2087.42} C_VEL
LIN {X 0,Y 705.1,Z 968.15,A -85,B 0,C 180,E1 -2089.036,E2 -2089.036} C_VEL
LIN {X 0,Y 705.546,Z 951.316,A -85,B 0,C 180,E1 -2090.715,E2 -2090.715} C_VEL
LIN {X 0,Y 706.047,Z 934.282,A -85,B 0,C 180,E1 -2092.217,E2 -2092.217} C_VEL
LIN {X 0,Y 706.624,Z 915.062,A -85,B 0,C 180,E1 -2093.695,E2 -2093.695} C_VEL
LIN {X 0,Y 707.258,Z 895.078,A -85,B 0,C 180,E1 -2095.051,E2 -2095.051} C_VEL
LIN {X 0,Y 707.906,Z 873.952,A -85,B 0,C 180,E1 -2096.283,E2 -2096.283} C_VEL
LIN {X 0,Y 708.585,Z 852.224,A -85,B 0,C 180,E1 -2097.389,E2 -2097.389} C_VEL
LIN {X 0,Y 709.16,Z 830.467,A -85,B 0,C 180,E1 -2098.324,E2 -2098.324} C_VEL
LIN {X 0,Y 709.784,Z 808.047,A -85,B 0,C 180,E1 -2099.142,E2 -2099.142} C_VEL
LIN {X 0,Y 710.27,Z 783.901,A -85,B 0,C 180,E1 -2099.855,E2 -2099.855} C_VEL
LIN {X 0,Y 710.715,Z 761.77,A -85,B 0,C 180,E1 -2100.371,E2 -2100.371} C_VEL
LIN {X 0,Y 711.1,Z 736.497,A -85,B 0,C 180,E1 -2100.8,E2 -2100.8} C_VEL
LIN {X 0,Y 712.564,Z 478.598,A -85,B 0,C 180,E1 -2103.764,E2 -2103.764} C_VEL
LIN {X 0,Y 713.042,Z 359.6,A -85,B 0,C 180,E1 -2105.161,E2 -2105.161} C_VEL
LIN {X 0,Y 709.992,Z 349.229,A -85,B 0,C 180,E1 -2105.46,E2 -2105.46} C_VEL
LIN {X 0,Y 709.099,Z 347.303,A -85,B 0,C 180,E1 -2105.548,E2 -2105.548} C_VEL
LIN {X 0,Y 704.3,Z 333.493,A -85,B 0,C 180,E1 -2106.937,E2 -2106.937} C_VEL
LIN {X 0,Y 704.296,Z 333.498,A -85,B 0,C 180,E1 -2110.025,E2 -2110.025} C_VEL
LIN {X 0,Y 704.274,Z 333.5,A -85,B 0,C 180,E1 -2112.656,E2 -2112.656} C_VEL
LIN {X 0,Y 704.345,Z 333.498,A -85,B 0,C 180,E1 -2115.566,E2 -2115.566} C_VEL
LIN {X 0,Y 704.273,Z 333.484,A -85,B 0,C 180,E1 -2118.469,E2 -2118.469} C_VEL
LIN {X 0,Y 704.298,Z 333.498,A -85,B 0,C 180,E1 -2121.133,E2 -2121.133} C_VEL
LIN {X 0,Y 704.301,Z 333.495,A -85,B 0,C 180,E1 -2124.203,E2 -2124.203} C_VEL
LIN {X 0,Y 704.273,Z 333.497,A -85,B 0,C 180,E1 -2126.893,E2 -2126.893} C_VEL
LIN {X 0,Y 704.347,Z 333.497,A -85,B 0,C 180,E1 -2129.738,E2 -2129.738} C_VEL
LIN {X 0,Y 704.278,Z 333.491,A -85,B 0,C 180,E1 -2132.613,E2 -2132.613} C_VEL
LIN {X 0,Y 704.277,Z 333.498,A -85,B 0,C 180,E1 -2135.15,E2 -2135.15} C_VEL
LIN {X 0,Y 704.343,Z 333.494,A -85,B 0,C 180,E1 -2138.077,E2 -2138.077} C_VEL
LIN {X 0,Y 704.274,Z 333.492,A -85,B 0,C 180,E1 -2140.855,E2 -2140.855} C_VEL
LIN {X 0,Y 704.295,Z 333.499,A -85,B 0,C 180,E1 -2143.504,E2 -2143.504} C_VEL
LIN {X 0,Y 704.295,Z 333.494,A -85,B 0,C 180,E1 -2146.62,E2 -2146.62} C_VEL
LIN {X 0,Y 704.272,Z 333.492,A -85,B 0,C 180,E1 -2149.281,E2 -2149.281} C_VEL
LIN {X 0,Y 704.344,Z 333.494,A -85,B 0,C 180,E1 -2152.167,E2 -2152.167} C_VEL
LIN {X 0,Y 704.275,Z 333.494,A -85,B 0,C 180,E1 -2155.032,E2 -2155.032} C_VEL
LIN {X 0,Y 704.284,Z 333.497,A -85,B 0,C 180,E1 -2157.64,E2 -2157.64} C_VEL
LIN {X 0,Y 704.321,Z 333.493,A -85,B 0,C 180,E1 -2160.651,E2 -2160.651} C_VEL
LIN {X 0,Y 704.269,Z 333.49,A -85,B 0,C 180,E1 -2163.337,E2 -2163.337} C_VEL
LIN {X 0,Y 704.313,Z 333.5,A -85,B 0,C 180,E1 -2166.03,E2 -2166.03} C_VEL
LIN {X 0,Y 704.288,Z 333.494,A -85,B 0,C 180,E1 -2169.067,E2 -2169.067} C_VEL
LIN {X 0,Y 704.272,Z 333.495,A -85,B 0,C 180,E1 -2171.631,E2 -2171.631} C_VEL
LIN {X 0,Y 704.346,Z 333.497,A -85,B 0,C 180,E1 -2174.495,E2 -2174.495} C_VEL
LIN {X 0,Y 704.277,Z 333.493,A -85,B 0,C 180,E1 -2177.346,E2 -2177.346} C_VEL
LIN {X 0,Y 704.278,Z 333.497,A -85,B 0,C 180,E1 -2179.922,E2 -2179.922} C_VEL
LIN {X 0,Y 704.341,Z 333.492,A -85,B 0,C 180,E1 -2182.891,E2 -2182.891} C_VEL
LIN {X 0,Y 704.271,Z 333.496,A -85,B 0,C 180,E1 -2185.66,E2 -2185.66} C_VEL
LIN {X 0,Y 704.301,Z 333.497,A -85,B 0,C 180,E1 -2188.332,E2 -2188.332} C_VEL
LIN {X 0,Y 704.286,Z 333.493,A -85,B 0,C 180,E1 -2191.433,E2 -2191.433} C_VEL
LIN {X 0,Y 704.271,Z 333.497,A -85,B 0,C 180,E1 -2194.013,E2 -2194.013} C_VEL
LIN {X 0,Y 704.345,Z 333.495,A -85,B 0,C 180,E1 -2196.905,E2 -2196.905} C_VEL
LIN {X 0,Y 704.272,Z 333.492,A -85,B 0,C 180,E1 -2199.818,E2 -2199.818} C_VEL
LIN {X 0,Y 704.285,Z 333.496,A -85,B 0,C 180,E1 -2202.417,E2 -2202.417} C_VEL
LIN {X 0,Y 704.312,Z 333.494,A -85,B 0,C 180,E1 -2205.467,E2 -2205.467} C_VEL
LIN {X 0,Y 704.27,Z 333.499,A -85,B 0,C 180,E1 -2208.142,E2 -2208.142} C_VEL
LIN {X 0,Y 704.337,Z 333.499,A -85,B 0,C 180,E1 -2210.961,E2 -2210.961} C_VEL
LIN {X 0,Y 710.716,Z 350.759,A -85,B 0,C 180,E1 -2212.673,E2 -2212.673} C_VEL
LIN {X 0,Y 710.234,Z 377.393,A -85,B 0,C 180,E1 -2214.576,E2 -2214.576} C_VEL
LIN {X 0,Y 713.272,Z 390.545,A -85,B 0,C 180,E1 -2214.908,E2 -2214.908} C_VEL
LIN {X 0,Y 711.768,Z 650.523,A -85,B 0,C 180,E1 -2217.91,E2 -2217.91} C_VEL
LIN {X 0,Y 711.095,Z 767.212,A -85,B 0,C 180,E1 -2219.254,E2 -2219.254} C_VEL
LIN {X 0,Y 710.676,Z 792.89,A -85,B 0,C 180,E1 -2219.697,E2 -2219.697} C_VEL
LIN {X 0,Y 710.261,Z 814.557,A -85,B 0,C 180,E1 -2220.208,E2 -2220.208} C_VEL
LIN {X 0,Y 709.764,Z 838.562,A -85,B 0,C 180,E1 -2220.92,E2 -2220.92} C_VEL
LIN {X 0,Y 709.159,Z 860.488,A -85,B 0,C 180,E1 -2221.722,E2 -2221.722} C_VEL
LIN {X 0,Y 708.561,Z 883.169,A -85,B 0,C 180,E1 -2222.701,E2 -2222.701} C_VEL
LIN {X 0,Y 707.877,Z 904.758,A -85,B 0,C 180,E1 -2223.806,E2 -2223.806} C_VEL
LIN {X 0,Y 707.237,Z 925.751,A -85,B 0,C 180,E1 -2225.038,E2 -2225.038} C_VEL
LIN {X 0,Y 706.621,Z 945.051,A -85,B 0,C 180,E1 -2226.349,E2 -2226.349} C_VEL
LIN {X 0,Y 706.067,Z 963.762,A -85,B 0,C 180,E1 -2227.783,E2 -2227.783} C_VEL
LIN {X 0,Y 705.558,Z 980.804,A -85,B 0,C 180,E1 -2229.282,E2 -2229.282} C_VEL
LIN {X 0,Y 705.129,Z 996.966,A -85,B 0,C 180,E1 -2230.879,E2 -2230.879} C_VEL
LIN {X 0,Y 704.773,Z 1011.223,A -85,B 0,C 180,E1 -2232.496,E2 -2232.496} C_VEL
LIN {X 0,Y 704.503,Z 1025.06,A -85,B 0,C 180,E1 -2234.271,E2 -2234.271} C_VEL
LIN {X 0,Y 704.267,Z 1036.797,A -85,B 0,C 180,E1 -2236.033,E2 -2236.033} C_VEL
LIN {X 0,Y 704.122,Z 1046.947,A -85,B 0,C 180,E1 -2237.785,E2 -2237.785} C_VEL
LIN {X 0,Y 704.017,Z 1056.538,A -85,B 0,C 180,E1 -2239.774,E2 -2239.774} C_VEL
LIN {X 0,Y 703.947,Z 1063.12,A -85,B 0,C 180,E1 -2241.423,E2 -2241.423} C_VEL
LIN {X 0,Y 703.913,Z 1069.451,A -85,B 0,C 180,E1 -2243.393,E2 -2243.393} C_VEL
LIN {X 0,Y 703.919,Z 1073.814,A -85,B 0,C 180,E1 -2245.274,E2 -2245.274} C_VEL
LIN {X 0,Y 703.909,Z 1076.797,A -85,B 0,C 180,E1 -2247.15,E2 -2247.15} C_VEL
LIN {X 0,Y 703.902,Z 1078.284,A -85,B 0,C 180,E1 -2249.186,E2 -2249.186} C_VEL
LIN {X 0,Y 703.907,Z 1078.262,A -85,B 0,C 180,E1 -2250.895,E2 -2250.895} C_VEL
LIN {X 0,Y 703.916,Z 1076.573,A -85,B 0,C 180,E1 -2253.013,E2 -2253.013} C_VEL
LIN {X 0,Y 703.919,Z 1073.655,A -85,B 0,C 180,E1 -2254.807,E2 -2254.807} C_VEL
LIN {X 0,Y 703.922,Z 1069.015,A -85,B 0,C 180,E1 -2256.771,E2 -2256.771} C_VEL
LIN {X 0,Y 703.945,Z 1062.816,A -85,B 0,C 180,E1 -2258.659,E2 -2258.659} C_VEL
LIN {X 0,Y 704.025,Z 1056.183,A -85,B 0,C 180,E1 -2260.309,E2 -2260.309} C_VEL
LIN {X 0,Y 704.135,Z 1046.031,A -85,B 0,C 180,E1 -2262.382,E2 -2262.382} C_VEL
LIN {X 0,Y 704.274,Z 1036.281,A -85,B 0,C 180,E1 -2264.05,E2 -2264.05} C_VEL
LIN {X 0,Y 704.516,Z 1023.805,A -85,B 0,C 180,E1 -2265.897,E2 -2265.897} C_VEL
LIN {X 0,Y 704.794,Z 1010.517,A -85,B 0,C 180,E1 -2267.589,E2 -2267.589} C_VEL
LIN {X 0,Y 705.159,Z 995.333,A -85,B 0,C 180,E1 -2269.292,E2 -2269.292} C_VEL
LIN {X 0,Y 705.592,Z 979.535,A -85,B 0,C 180,E1 -2270.836,E2 -2270.836} C_VEL
LIN {X 0,Y 706.116,Z 961.608,A -85,B 0,C 180,E1 -2272.39,E2 -2272.39} C_VEL
LIN {X 0,Y 706.659,Z 944.007,A -85,B 0,C 180,E1 -2273.726,E2 -2273.726} C_VEL
LIN {X 0,Y 707.287,Z 923.623,A -85,B 0,C 180,E1 -2275.094,E2 -2275.094} C_VEL
LIN {X 0,Y 707.908,Z 903.834,A -85,B 0,C 180,E1 -2276.244,E2 -2276.244} C_VEL
LIN {X 0,Y 708.586,Z 882.241,A -85,B 0,C 180,E1 -2277.343,E2 -2277.343} C_VEL
LIN {X 0,Y 709.195,Z 859.367,A -85,B 0,C 180,E1 -2278.322,E2 -2278.322} C_VEL
LIN {X 0,Y 709.833,Z 836.517,A -85,B 0,C 180,E1 -2279.149,E2 -2279.149} C_VEL
LIN {X 0,Y 710.283,Z 812.684,A -85,B 0,C 180,E1 -2279.842,E2 -2279.842} C_VEL
LIN {X 0,Y 710.8,Z 788.99,A -85,B 0,C 180,E1 -2280.384,E2 -2280.384} C_VEL
LIN {X 0,Y 711.11,Z 764.773,A -85,B 0,C 180,E1 -2280.778,E2 -2280.778} C_VEL
LIN {X 0,Y 712.515,Z 513.855,A -85,B 0,C 180,E1 -2283.659,E2 -2283.659} C_VEL
LIN {X 0,Y 713.088,Z 388.851,A -85,B 0,C 180,E1 -2285.122,E2 -2285.122} C_VEL
LIN {X 0,Y 710.16,Z 376.686,A -85,B 0,C 180,E1 -2285.457,E2 -2285.457} C_VEL
LIN {X 0,Y 710.659,Z 350.511,A -85,B 0,C 180,E1 -2287.349,E2 -2287.349} C_VEL
LIN {X 0,Y 704.336,Z 333.49,A -85,B 0,C 180,E1 -2289.038,E2 -2289.038} C_VEL
LIN {X 0,Y 704.271,Z 333.499,A -85,B 0,C 180,E1 -2291.858,E2 -2291.858} C_VEL
LIN {X 0,Y 704.313,Z 333.495,A -85,B 0,C 180,E1 -2294.547,E2 -2294.547} C_VEL
LIN {X 0,Y 704.287,Z 333.498,A -85,B 0,C 180,E1 -2297.595,E2 -2297.595} C_VEL
LIN {X 0,Y 704.273,Z 333.494,A -85,B 0,C 180,E1 -2300.185,E2 -2300.185} C_VEL
LIN {X 0,Y 704.345,Z 333.489,A -85,B 0,C 180,E1 -2303.057,E2 -2303.057} C_VEL
LIN {X 0,Y 704.277,Z 333.495,A -85,B 0,C 180,E1 -2305.889,E2 -2305.889} C_VEL
LIN {X 0,Y 704.283,Z 333.492,A -85,B 0,C 180,E1 -2308.502,E2 -2308.502} C_VEL
LIN {X 0,Y 704.326,Z 333.495,A -85,B 0,C 180,E1 -2311.51,E2 -2311.51} C_VEL
LIN {X 0,Y 704.272,Z 333.496,A -85,B 0,C 180,E1 -2314.25,E2 -2314.25} C_VEL
LIN {X 0,Y 704.328,Z 333.49,A -85,B 0,C 180,E1 -2317.02,E2 -2317.02} C_VEL
LIN {X 0,Y 704.284,Z 333.496,A -85,B 0,C 180,E1 -2320.027,E2 -2320.027} C_VEL
LIN {X 0,Y 704.28,Z 333.494,A -85,B 0,C 180,E1 -2322.654,E2 -2322.654} C_VEL
LIN {X 0,Y 704.344,Z 333.497,A -85,B 0,C 180,E1 -2325.615,E2 -2325.615} C_VEL
LIN {X 0,Y 704.274,Z 333.493,A -85,B 0,C 180,E1 -2328.452,E2 -2328.452} C_VEL
LIN {X 0,Y 704.317,Z 333.493,A -85,B 0,C 180,E1 -2331.18,E2 -2331.18} C_VEL
LIN {X 0,Y 704.29,Z 333.499,A -85,B 0,C 180,E1 -2334.215,E2 -2334.215} C_VEL
LIN {X 0,Y 704.277,Z 333.492,A -85,B 0,C 180,E1 -2336.826,E2 -2336.826} C_VEL
LIN {X 0,Y 704.346,Z 333.496,A -85,B 0,C 180,E1 -2339.756,E2 -2339.756} C_VEL
LIN {X 0,Y 704.276,Z 333.494,A -85,B 0,C 180,E1 -2342.604,E2 -2342.604} C_VEL
LIN {X 0,Y 704.303,Z 333.493,A -85,B 0,C 180,E1 -2345.295,E2 -2345.295} C_VEL
LIN {X 0,Y 704.297,Z 333.499,A -85,B 0,C 180,E1 -2348.409,E2 -2348.409} C_VEL
LIN {X 0,Y 704.277,Z 333.491,A -85,B 0,C 180,E1 -2351.05,E2 -2351.05} C_VEL
LIN {X 0,Y 704.345,Z 333.496,A -85,B 0,C 180,E1 -2353.965,E2 -2353.965} C_VEL
LIN {X 0,Y 704.279,Z 333.496,A -85,B 0,C 180,E1 -2356.836,E2 -2356.836} C_VEL
LIN {X 0,Y 704.299,Z 333.492,A -85,B 0,C 180,E1 -2359.494,E2 -2359.494} C_VEL
LIN {X 0,Y 704.338,Z 333.491,A -85,B 0,C 180,E1 -2361.85,E2 -2361.85} C_VEL
LIN {X 0,Y 703.383,Z 333.619,A -85,B 0,C 180,E1 -2362.476,E2 -2362.476} C_VEL
LIN {X 0,Y 696.932,Z 334.423,A -85,B 0,C 180,E1 -2364.231,E2 -2364.231} C_VEL
LIN {X 0,Y 696.359,Z 334.487,A -85,B 0,C 180,E1 -2364.688,E2 -2364.688} C_VEL
LIN {X 0,Y 696.343,Z 334.481,A -85,B 0,C 180,E1 -2367.355,E2 -2367.355} C_VEL
LIN {X 0,Y 696.407,Z 334.486,A -85,B 0,C 180,E1 -2370.263,E2 -2370.263} C_VEL
LIN {X 0,Y 696.341,Z 334.486,A -85,B 0,C 180,E1 -2373.168,E2 -2373.168} C_VEL
LIN {X 0,Y 696.384,Z 334.481,A -85,B 0,C 180,E1 -2375.963,E2 -2375.963} C_VEL
LIN {X 0,Y 696.353,Z 334.488,A -85,B 0,C 180,E1 -2379.03,E2 -2379.03} C_VEL
LIN {X 0,Y 696.349,Z 334.485,A -85,B 0,C 180,E1 -2381.697,E2 -2381.697} C_VEL
LIN {X 0,Y 696.398,Z 334.486,A -85,B 0,C 180,E1 -2384.712,E2 -2384.712} C_VEL
LIN {X 0,Y 696.341,Z 334.488,A -85,B 0,C 180,E1 -2387.555,E2 -2387.555} C_VEL
LIN {X 0,Y 696.404,Z 334.486,A -85,B 0,C 180,E1 -2390.395,E2 -2390.395} C_VEL
LIN {X 0,Y 696.428,Z 334.656,A -85,B 0,C 180,E1 -2392.751,E2 -2392.751} C_VEL
LIN {X 0,Y 701.14,Z 347.989,A -85,B 0,C 180,E1 -2394.098,E2 -2394.098} C_VEL
LIN {X 0,Y 704.659,Z 354.748,A -85,B 0,C 180,E1 -2394.389,E2 -2394.389} C_VEL
LIN {X 0,Y 706.664,Z 362.972,A -85,B 0,C 180,E1 -2394.606,E2 -2394.606} C_VEL
LIN {X 0,Y 705.107,Z 602.463,A -85,B 0,C 180,E1 -2397.401,E2 -2397.401} C_VEL
LIN {X 0,Y 704.211,Z 737.148,A -85,B 0,C 180,E1 -2398.965,E2 -2398.965} C_VEL
LIN {X 0,Y 703.748,Z 762.739,A -85,B 0,C 180,E1 -2399.409,E2 -2399.409} C_VEL
LIN {X 0,Y 703.256,Z 784.537,A -85,B 0,C 180,E1 -2399.925,E2 -2399.925} C_VEL
LIN {X 0,Y 702.684,Z 808.612,A -85,B 0,C 180,E1 -2400.646,E2 -2400.646} C_VEL
LIN {X 0,Y 702.042,Z 829.399,A -85,B 0,C 180,E1 -2401.409,E2 -2401.409} C_VEL
LIN {X 0,Y 701.346,Z 851.276,A -85,B 0,C 180,E1 -2402.351,E2 -2402.351} C_VEL
LIN {X 0,Y 700.587,Z 873.151,A -85,B 0,C 180,E1 -2403.467,E2 -2403.467} C_VEL
LIN {X 0,Y 699.872,Z 892.904,A -85,B 0,C 180,E1 -2404.621,E2 -2404.621} C_VEL
LIN {X 0,Y 699.15,Z 912.981,A -85,B 0,C 180,E1 -2405.973,E2 -2405.973} C_VEL
LIN {X 0,Y 698.518,Z 930.639,A -85,B 0,C 180,E1 -2407.32,E2 -2407.32} C_VEL
LIN {X 0,Y 697.901,Z 949.06,A -85,B 0,C 180,E1 -2408.924,E2 -2408.924} C_VEL
LIN {X 0,Y 697.39,Z 964.894,A -85,B 0,C 180,E1 -2410.484,E2 -2410.484} C_VEL
LIN {X 0,Y 696.961,Z 980.15,A -85,B 0,C 180,E1 -2412.207,E2 -2412.207} C_VEL
LIN {X 0,Y 696.62,Z 993.469,A -85,B 0,C 180,E1 -2413.918,E2 -2413.918} C_VEL
LIN {X 0,Y 696.353,Z 1006.007,A -85,B 0,C 180,E1 -2415.786,E2 -2415.786} C_VEL
LIN {X 0,Y 696.186,Z 1015.785,A -85,B 0,C 180,E1 -2417.475,E2 -2417.475} C_VEL
LIN {X 0,Y 696.048,Z 1025.993,A -85,B 0,C 180,E1 -2419.572,E2 -2419.572} C_VEL
LIN {X 0,Y 695.953,Z 1032.956,A -85,B 0,C 180,E1 -2421.324,E2 -2421.324} C_VEL
LIN {X 0,Y 695.936,Z 1039.125,A -85,B 0,C 180,E1 -2423.234,E2 -2423.234} C_VEL
LIN {X 0,Y 695.908,Z 1043.728,A -85,B 0,C 180,E1 -2425.22,E2 -2425.22} C_VEL
LIN {X 0,Y 695.912,Z 1046.511,A -85,B 0,C 180,E1 -2426.953,E2 -2426.953} C_VEL
LIN {X 0,Y 695.907,Z 1048.249,A -85,B 0,C 180,E1 -2429.094,E2 -2429.094} C_VEL
LIN {X 0,Y 695.902,Z 1048.296,A -85,B 0,C 180,E1 -2430.823,E2 -2430.823} C_VEL
LIN {X 0,Y 695.899,Z 1046.971,A -85,B 0,C 180,E1 -2432.8,E2 -2432.8} C_VEL
LIN {X 0,Y 695.916,Z 1044.059,A -85,B 0,C 180,E1 -2434.698,E2 -2434.698} C_VEL
LIN {X 0,Y 695.919,Z 1040.183,A -85,B 0,C 180,E1 -2436.435,E2 -2436.435} C_VEL
LIN {X 0,Y 695.954,Z 1033.89,A -85,B 0,C 180,E1 -2438.51,E2 -2438.51} C_VEL
LIN {X 0,Y 696.032,Z 1027.085,A -85,B 0,C 180,E1 -2440.261,E2 -2440.261} C_VEL
LIN {X 0,Y 696.153,Z 1018.102,A -85,B 0,C 180,E1 -2442.189,E2 -2442.189} C_VEL
LIN {X 0,Y 696.323,Z 1007.594,A -85,B 0,C 180,E1 -2444.045,E2 -2444.045} C_VEL
LIN {X 0,Y 696.572,Z 995.948,A -85,B 0,C 180,E1 -2445.827,E2 -2445.827} C_VEL
LIN {X 0,Y 696.894,Z 982.299,A -85,B 0,C 180,E1 -2447.622,E2 -2447.622} C_VEL
LIN {X 0,Y 697.295,Z 968.146,A -85,B 0,C 180,E1 -2449.257,E2 -2449.257} C_VEL
LIN {X 0,Y 697.808,Z 951.862,A -85,B 0,C 180,E1 -2450.903,E2 -2450.903} C_VEL
LIN {X 0,Y 698.361,Z 935.289,A -85,B 0,C 180,E1 -2452.386,E2 -2452.386} C_VEL
LIN {X 0,Y 699.032,Z 916.263,A -85,B 0,C 180,E1 -2453.879,E2 -2453.879} C_VEL
LIN {X 0,Y 699.697,Z 897.748,A -85,B 0,C 180,E1 -2455.159,E2 -2455.159} C_VEL
LIN {X 0,Y 700.465,Z 876.355,A -85,B 0,C 180,E1 -2456.447,E2 -2456.447} C_VEL
LIN {X 0,Y 701.167,Z 856.657,A -85,B 0,C 180,E1 -2457.477,E2 -2457.477} C_VEL
LIN {X 0,Y 701.929,Z 832.695,A -85,B 0,C 180,E1 -2458.549,E2 -2458.549} C_VEL
LIN {X 0,Y 702.549,Z 812.364,A -85,B 0,C 180,E1 -2459.314,E2 -2459.314} C_VEL
LIN {X 0,Y 703.221,Z 787.502,A -85,B 0,C 180,E1 -2460.086,E2 -2460.086} C_VEL
LIN {X 0,Y 703.676,Z 765.394,A -85,B 0,C 180,E1 -2460.625,E2 -2460.625} C_VEL
LIN {X 0,Y 704.188,Z 740.796,A -85,B 0,C 180,E1 -2461.076,E2 -2461.076} C_VEL
LIN {X 0,Y 704.537,Z 693.711,A -85,B 0,C 180,E1 -2461.643,E2 -2461.643} C_VEL
LIN {X 0,Y 706.175,Z 439.974,A -85,B 0,C 180,E1 -2464.576,E2 -2464.576} C_VEL
LIN {X 0,Y 706.502,Z 361.588,A -85,B 0,C 180,E1 -2465.51,E2 -2465.51} C_VEL
LIN {X 0,Y 703.94,Z 352.965,A -85,B 0,C 180,E1 -2465.765,E2 -2465.765} C_VEL
LIN {X 0,Y 700.898,Z 347.486,A -85,B 0,C 180,E1 -2466.014,E2 -2466.014} C_VEL
LIN {X 0,Y 696.403,Z 334.475,A -85,B 0,C 180,E1 -2467.359,E2 -2467.359} C_VEL
LIN {X 0,Y 696.339,Z 334.489,A -85,B 0,C 180,E1 -2470.253,E2 -2470.253} C_VEL
LIN {X 0,Y 696.348,Z 334.49,A -85,B 0,C 180,E1 -2472.892,E2 -2472.892} C_VEL
LIN {X 0,Y 696.371,Z 334.486,A -85,B 0,C 180,E1 -2476.002,E2 -2476.002} C_VEL
LIN {X 0,Y 696.332,Z 334.473,A -85,B 0,C 180,E1 -2478.677,E2 -2478.677} C_VEL
LIN {X 0,Y 696.402,Z 334.488,A -85,B 0,C 180,E1 -2481.491,E2 -2481.491} C_VEL
LIN {X 0,Y 696.341,Z 334.485,A -85,B 0,C 180,E1 -2484.44,E2 -2484.44} C_VEL
LIN {X 0,Y 696.341,Z 334.486,A -85,B 0,C 180,E1 -2487.029,E2 -2487.029} C_VEL
LIN {X 0,Y 696.401,Z 334.482,A -85,B 0,C 180,E1 -2490.022,E2 -2490.022} C_VEL
LIN {X 0,Y 696.333,Z 334.481,A -85,B 0,C 180,E1 -2492.83,E2 -2492.83} C_VEL
LIN {X 0,Y 696.381,Z 334.488,A -85,B 0,C 180,E1 -2495.574,E2 -2495.574} C_VEL
LIN {X 0,Y 696.345,Z 334.484,A -85,B 0,C 180,E1 -2498.609,E2 -2498.609} C_VEL
LIN {X 0,Y 696.339,Z 334.483,A -85,B 0,C 180,E1 -2501.237,E2 -2501.237} C_VEL
LIN {X 0,Y 696.404,Z 334.477,A -85,B 0,C 180,E1 -2504.169,E2 -2504.169} C_VEL
LIN {X 0,Y 696.334,Z 334.485,A -85,B 0,C 180,E1 -2506.971,E2 -2506.971} C_VEL
LIN {X 0,Y 696.36,Z 334.482,A -85,B 0,C 180,E1 -2509.66,E2 -2509.66} C_VEL
LIN {X 0,Y 696.354,Z 334.48,A -85,B 0,C 180,E1 -2512.741,E2 -2512.741} C_VEL
LIN {X 0,Y 696.334,Z 334.485,A -85,B 0,C 180,E1 -2515.388,E2 -2515.388} C_VEL
LIN {X 0,Y 696.406,Z 334.48,A -85,B 0,C 180,E1 -2518.272,E2 -2518.272} C_VEL
LIN {X 0,Y 696.336,Z 334.485,A -85,B 0,C 180,E1 -2521.152,E2 -2521.152} C_VEL
LIN {X 0,Y 696.349,Z 334.481,A -85,B 0,C 180,E1 -2523.787,E2 -2523.787} C_VEL
LIN {X 0,Y 696.359,Z 334.479,A -85,B 0,C 180,E1 -2526.928,E2 -2526.928} C_VEL
LIN {X 0,Y 696.333,Z 334.486,A -85,B 0,C 180,E1 -2529.588,E2 -2529.588} C_VEL
LIN {X 0,Y 696.405,Z 334.482,A -85,B 0,C 180,E1 -2532.489,E2 -2532.489} C_VEL
LIN {X 0,Y 696.335,Z 334.484,A -85,B 0,C 180,E1 -2535.406,E2 -2535.406} C_VEL
LIN {X 0,Y 696.345,Z 334.485,A -85,B 0,C 180,E1 -2537.982,E2 -2537.982} C_VEL
LIN {X 0,Y 696.374,Z 334.48,A -85,B 0,C 180,E1 -2541.044,E2 -2541.044} C_VEL
LIN {X 0,Y 696.332,Z 334.484,A -85,B 0,C 180,E1 -2543.707,E2 -2543.707} C_VEL
LIN {X 0,Y 696.38,Z 334.488,A -85,B 0,C 180,E1 -2546.431,E2 -2546.431} C_VEL
LIN {X 0,Y 696.349,Z 334.485,A -85,B 0,C 180,E1 -2549.412,E2 -2549.412} C_VEL
LIN {X 0,Y 696.332,Z 334.485,A -85,B 0,C 180,E1 -2551.996,E2 -2551.996} C_VEL
LIN {X 0,Y 696.406,Z 334.485,A -85,B 0,C 180,E1 -2554.851,E2 -2554.851} C_VEL
LIN {X 0,Y 696.337,Z 334.485,A -85,B 0,C 180,E1 -2557.713,E2 -2557.713} C_VEL
LIN {X 0,Y 696.343,Z 334.483,A -85,B 0,C 180,E1 -2560.317,E2 -2560.317} C_VEL
LIN {X 0,Y 696.386,Z 334.482,A -85,B 0,C 180,E1 -2563.34,E2 -2563.34} C_VEL
LIN {X 0,Y 696.332,Z 334.486,A -85,B 0,C 180,E1 -2566.124,E2 -2566.124} C_VEL
LIN {X 0,Y 696.404,Z 334.485,A -85,B 0,C 180,E1 -2568.993,E2 -2568.993} C_VEL
LIN {X 0,Y 696.357,Z 334.562,A -85,B 0,C 180,E1 -2570.559,E2 -2570.559} C_VEL
LIN {X 0,Y 703.698,Z 354.082,A -85,B 0,C 180,E1 -2572.493,E2 -2572.493} C_VEL
LIN {X 0,Y 703.259,Z 377.512,A -85,B 0,C 180,E1 -2574.173,E2 -2574.173} C_VEL
LIN {X 0,Y 706.71,Z 392.225,A -85,B 0,C 180,E1 -2574.554,E2 -2574.554} C_VEL
LIN {X 0,Y 704.975,Z 652.28,A -85,B 0,C 180,E1 -2577.584,E2 -2577.584} C_VEL
LIN {X 0,Y 704.208,Z 767.352,A -85,B 0,C 180,E1 -2578.922,E2 -2578.922} C_VEL
LIN {X 0,Y 703.74,Z 793.019,A -85,B 0,C 180,E1 -2579.37,E2 -2579.37} C_VEL
LIN {X 0,Y 703.252,Z 814.776,A -85,B 0,C 180,E1 -2579.886,E2 -2579.886} C_VEL
LIN {X 0,Y 702.642,Z 839.843,A -85,B 0,C 180,E1 -2580.644,E2 -2580.644} C_VEL
LIN {X 0,Y 702.006,Z 860.487,A -85,B 0,C 180,E1 -2581.408,E2 -2581.408} C_VEL
LIN {X 0,Y 701.296,Z 883.165,A -85,B 0,C 180,E1 -2582.395,E2 -2582.395} C_VEL
LIN {X 0,Y 700.533,Z 904.595,A -85,B 0,C 180,E1 -2583.501,E2 -2583.501} C_VEL
LIN {X 0,Y 699.772,Z 925.765,A -85,B 0,C 180,E1 -2584.754,E2 -2584.754} C_VEL
LIN {X 0,Y 699.086,Z 944.774,A -85,B 0,C 180,E1 -2586.058,E2 -2586.058} C_VEL
LIN {X 0,Y 698.419,Z 963.761,A -85,B 0,C 180,E1 -2587.527,E2 -2587.527} C_VEL
LIN {X 0,Y 697.847,Z 980.462,A -85,B 0,C 180,E1 -2589.01,E2 -2589.01} C_VEL
LIN {X 0,Y 697.33,Z 996.968,A -85,B 0,C 180,E1 -2590.657,E2 -2590.657} C_VEL
LIN {X 0,Y 696.908,Z 1011.933,A -85,B 0,C 180,E1 -2592.378,E2 -2592.378} C_VEL
LIN {X 0,Y 696.571,Z 1026.223,A -85,B 0,C 180,E1 -2594.258,E2 -2594.258} C_VEL
LIN {X 0,Y 696.32,Z 1037.318,A -85,B 0,C 180,E1 -2595.955,E2 -2595.955} C_VEL
LIN {X 0,Y 696.148,Z 1047.863,A -85,B 0,C 180,E1 -2597.811,E2 -2597.811} C_VEL
LIN {X 0,Y 696.032,Z 1056.95,A -85,B 0,C 180,E1 -2599.752,E2 -2599.752} C_VEL
LIN {X 0,Y 695.955,Z 1063.727,A -85,B 0,C 180,E1 -2601.49,E2 -2601.49} C_VEL
LIN {X 0,Y 695.914,Z 1070.07,A -85,B 0,C 180,E1 -2603.565,E2 -2603.565} C_VEL
LIN {X 0,Y 695.919,Z 1073.973,A -85,B 0,C 180,E1 -2605.302,E2 -2605.302} C_VEL
LIN {X 0,Y 695.907,Z 1077.017,A -85,B 0,C 180,E1 -2607.282,E2 -2607.282} C_VEL
LIN {X 0,Y 695.897,Z 1078.306,A -85,B 0,C 180,E1 -2609.259,E2 -2609.259} C_VEL
LIN {X 0,Y 695.914,Z 1078.239,A -85,B 0,C 180,E1 -2610.988,E2 -2610.988} C_VEL
LIN {X 0,Y 695.917,Z 1076.46,A -85,B 0,C 180,E1 -2613.13,E2 -2613.13} C_VEL
LIN {X 0,Y 695.92,Z 1073.497,A -85,B 0,C 180,E1 -2614.945,E2 -2614.945} C_VEL
LIN {X 0,Y 695.946,Z 1068.507,A -85,B 0,C 180,E1 -2617.015,E2 -2617.015} C_VEL
LIN {X 0,Y 695.954,Z 1062.816,A -85,B 0,C 180,E1 -2618.76,E2 -2618.76} C_VEL
LIN {X 0,Y 696.049,Z 1055.829,A -85,B 0,C 180,E1 -2620.512,E2 -2620.512} C_VEL
LIN {X 0,Y 696.176,Z 1046.03,A -85,B 0,C 180,E1 -2622.525,E2 -2622.525} C_VEL
LIN {X 0,Y 696.344,Z 1036.084,A -85,B 0,C 180,E1 -2624.246,E2 -2624.246} C_VEL
LIN {X 0,Y 696.624,Z 1022.856,A -85,B 0,C 180,E1 -2626.21,E2 -2626.21} C_VEL
LIN {X 0,Y 696.975,Z 1009.811,A -85,B 0,C 180,E1 -2627.879,E2 -2627.879} C_VEL
LIN {X 0,Y 697.431,Z 993.64,A -85,B 0,C 180,E1 -2629.689,E2 -2629.689} C_VEL
LIN {X 0,Y 697.91,Z 978.606,A -85,B 0,C 180,E1 -2631.164,E2 -2631.164} C_VEL
LIN {X 0,Y 698.56,Z 959.399,A -85,B 0,C 180,E1 -2632.824,E2 -2632.824} C_VEL
LIN {X 0,Y 699.194,Z 941.727,A -85,B 0,C 180,E1 -2634.163,E2 -2634.163} C_VEL
LIN {X 0,Y 699.978,Z 919.991,A -85,B 0,C 180,E1 -2635.601,E2 -2635.601} C_VEL
LIN {X 0,Y 700.677,Z 900.705,A -85,B 0,C 180,E1 -2636.713,E2 -2636.713} C_VEL
LIN {X 0,Y 701.468,Z 877.276,A -85,B 0,C 180,E1 -2637.875,E2 -2637.875} C_VEL
LIN {X 0,Y 702.12,Z 857.102,A -85,B 0,C 180,E1 -2638.727,E2 -2638.727} C_VEL
LIN {X 0,Y 702.823,Z 832.979,A -85,B 0,C 180,E1 -2639.582,E2 -2639.582} C_VEL
LIN {X 0,Y 703.338,Z 811.077,A -85,B 0,C 180,E1 -2640.21,E2 -2640.21} C_VEL
LIN {X 0,Y 703.916,Z 786.571,A -85,B 0,C 180,E1 -2640.761,E2 -2640.761} C_VEL
LIN {X 0,Y 704.235,Z 763.542,A -85,B 0,C 180,E1 -2641.129,E2 -2641.129} C_VEL
LIN {X 0,Y 705.84,Z 515.509,A -85,B 0,C 180,E1 -2644,E2 -2644} C_VEL
LIN {X 0,Y 706.538,Z 390.715,A -85,B 0,C 180,E1 -2645.474,E2 -2645.474} C_VEL
LIN {X 0,Y 703.158,Z 376.686,A -85,B 0,C 180,E1 -2645.864,E2 -2645.864} C_VEL
LIN {X 0,Y 703.62,Z 353.737,A -85,B 0,C 180,E1 -2647.537,E2 -2647.537} C_VEL
LIN {X 0,Y 696.347,Z 334.491,A -85,B 0,C 180,E1 -2649.462,E2 -2649.462} C_VEL
LIN {X 0,Y 696.335,Z 334.487,A -85,B 0,C 180,E1 -2652.065,E2 -2652.065} C_VEL
LIN {X 0,Y 696.407,Z 334.487,A -85,B 0,C 180,E1 -2654.943,E2 -2654.943} C_VEL
LIN {X 0,Y 696.336,Z 334.486,A -85,B 0,C 180,E1 -2657.811,E2 -2657.811} C_VEL
LIN {X 0,Y 696.352,Z 334.482,A -85,B 0,C 180,E1 -2660.451,E2 -2660.451} C_VEL
LIN {X 0,Y 696.364,Z 334.469,A -85,B 0,C 180,E1 -2663.526,E2 -2663.526} C_VEL
LIN {X 0,Y 696.334,Z 334.482,A -85,B 0,C 180,E1 -2666.243,E2 -2666.243} C_VEL
LIN {X 0,Y 696.407,Z 334.48,A -85,B 0,C 180,E1 -2669.164,E2 -2669.164} C_VEL
LIN {X 0,Y 696.337,Z 334.481,A -85,B 0,C 180,E1 -2672.018,E2 -2672.018} C_VEL
LIN {X 0,Y 696.351,Z 334.483,A -85,B 0,C 180,E1 -2674.666,E2 -2674.666} C_VEL
LIN {X 0,Y 696.364,Z 334.488,A -85,B 0,C 180,E1 -2677.813,E2 -2677.813} C_VEL
LIN {X 0,Y 696.334,Z 334.483,A -85,B 0,C 180,E1 -2680.453,E2 -2680.453} C_VEL
LIN {X 0,Y 696.404,Z 334.482,A -85,B 0,C 180,E1 -2683.312,E2 -2683.312} C_VEL
LIN {X 0,Y 696.342,Z 334.487,A -85,B 0,C 180,E1 -2686.21,E2 -2686.21} C_VEL
LIN {X 0,Y 696.346,Z 334.479,A -85,B 0,C 180,E1 -2688.823,E2 -2688.823} C_VEL
LIN {X 0,Y 696.393,Z 334.482,A -85,B 0,C 180,E1 -2691.828,E2 -2691.828} C_VEL
LIN {X 0,Y 696.337,Z 334.486,A -85,B 0,C 180,E1 -2694.562,E2 -2694.562} C_VEL
LIN {X 0,Y 696.387,Z 334.478,A -85,B 0,C 180,E1 -2697.367,E2 -2697.367} C_VEL
LIN {X 0,Y 696.346,Z 334.485,A -85,B 0,C 180,E1 -2700.411,E2 -2700.411} C_VEL
LIN {X 0,Y 696.346,Z 334.481,A -85,B 0,C 180,E1 -2703.046,E2 -2703.046} C_VEL
LIN {X 0,Y 696.39,Z 334.482,A -85,B 0,C 180,E1 -2706.099,E2 -2706.099} C_VEL
LIN {X 0,Y 696.337,Z 334.485,A -85,B 0,C 180,E1 -2708.838,E2 -2708.838} C_VEL
LIN {X 0,Y 696.396,Z 334.476,A -85,B 0,C 180,E1 -2711.68,E2 -2711.68} C_VEL
LIN {X 0,Y 696.348,Z 334.484,A -85,B 0,C 180,E1 -2714.639,E2 -2714.639} C_VEL
LIN {X 0,Y 696.348,Z 334.483,A -85,B 0,C 180,E1 -2717.292,E2 -2717.292} C_VEL
LIN {X 0,Y 696.393,Z 334.484,A -85,B 0,C 180,E1 -2720.333,E2 -2720.333} C_VEL
LIN {X 0,Y 696.339,Z 334.483,A -85,B 0,C 180,E1 -2723.08,E2 -2723.08} C_VEL
LIN {X 0,Y 696.359,Z 334.487,A -85,B 0,C 180,E1 -2724.688,E2 -2724.688} C_VEL
LIN {X 0,Y 695.323,Z 334.614,A -85,B 0,C 180,E1 -2725.322,E2 -2725.322} C_VEL
LIN {X 0,Y 688.917,Z 335.408,A -85,B 0,C 180,E1 -2727.098,E2 -2727.098} C_VEL
LIN {X 0,Y 688.416,Z 335.469,A -85,B 0,C 180,E1 -2727.56,E2 -2727.56} C_VEL
LIN {X 0,Y 688.431,Z 335.472,A -85,B 0,C 180,E1 -2730.703,E2 -2730.703} C_VEL
LIN {X 0,Y 688.403,Z 335.473,A -85,B 0,C 180,E1 -2733.401,E2 -2733.401} C_VEL
LIN {X 0,Y 688.466,Z 335.473,A -85,B 0,C 180,E1 -2736.339,E2 -2736.339} C_VEL
LIN {X 0,Y 688.403,Z 335.475,A -85,B 0,C 180,E1 -2739.27,E2 -2739.27} C_VEL
LIN {X 0,Y 688.448,Z 335.472,A -85,B 0,C 180,E1 -2742.084,E2 -2742.084} C_VEL
LIN {X 0,Y 688.414,Z 335.477,A -85,B 0,C 180,E1 -2745.138,E2 -2745.138} C_VEL
LIN {X 0,Y 688.413,Z 335.475,A -85,B 0,C 180,E1 -2747.853,E2 -2747.853} C_VEL
LIN {X 0,Y 688.449,Z 335.479,A -85,B 0,C 180,E1 -2750.925,E2 -2750.925} C_VEL
LIN {X 0,Y 688.479,Z 335.641,A -85,B 0,C 180,E1 -2752.307,E2 -2752.307} C_VEL
LIN {X 0,Y 692.877,Z 347.993,A -85,B 0,C 180,E1 -2753.6,E2 -2753.6} C_VEL
LIN {X 0,Y 698.653,Z 358.553,A -85,B 0,C 180,E1 -2754.082,E2 -2754.082} C_VEL
LIN {X 0,Y 700.126,Z 364.942,A -85,B 0,C 180,E1 -2754.249,E2 -2754.249} C_VEL
LIN {X 0,Y 698.349,Z 604.93,A -85,B 0,C 180,E1 -2757.075,E2 -2757.075} C_VEL
LIN {X 0,Y 697.35,Z 737.299,A -85,B 0,C 180,E1 -2758.626,E2 -2758.626} C_VEL
LIN {X 0,Y 696.841,Z 762.764,A -85,B 0,C 180,E1 -2759.072,E2 -2759.072} C_VEL
LIN {X 0,Y 696.276,Z 784.557,A -85,B 0,C 180,E1 -2759.591,E2 -2759.591} C_VEL
LIN {X 0,Y 695.631,Z 808.625,A -85,B 0,C 180,E1 -2760.319,E2 -2760.319} C_VEL
LIN {X 0,Y 694.91,Z 829.409,A -85,B 0,C 180,E1 -2761.088,E2 -2761.088} C_VEL
LIN {X 0,Y 694.12,Z 851.194,A -85,B 0,C 180,E1 -2762.033,E2 -2762.033} C_VEL
LIN {X 0,Y 693.259,Z 873.157,A -85,B 0,C 180,E1 -2763.164,E2 -2763.164} C_VEL
LIN {X 0,Y 692.459,Z 892.916,A -85,B 0,C 180,E1 -2764.33,E2 -2764.33} C_VEL
LIN {X 0,Y 691.609,Z 913.235,A -85,B 0,C 180,E1 -2765.713,E2 -2765.713} C_VEL
LIN {X 0,Y 690.884,Z 931.387,A -85,B 0,C 180,E1 -2767.115,E2 -2767.115} C_VEL
LIN {X 0,Y 690.199,Z 949.066,A -85,B 0,C 180,E1 -2768.677,E2 -2768.677} C_VEL
LIN {X 0,Y 689.626,Z 964.898,A -85,B 0,C 180,E1 -2770.256,E2 -2770.256} C_VEL
LIN {X 0,Y 689.123,Z 980.156,A -85,B 0,C 180,E1 -2771.998,E2 -2771.998} C_VEL
LIN {X 0,Y 688.741,Z 992.989,A -85,B 0,C 180,E1 -2773.663,E2 -2773.663} C_VEL
LIN {X 0,Y 688.422,Z 1006.173,A -85,B 0,C 180,E1 -2775.646,E2 -2775.646} C_VEL
LIN {X 0,Y 688.23,Z 1015.787,A -85,B 0,C 180,E1 -2777.327,E2 -2777.327} C_VEL
LIN {X 0,Y 688.063,Z 1025.641,A -85,B 0,C 180,E1 -2779.365,E2 -2779.365} C_VEL
LIN {X 0,Y 687.969,Z 1032.654,A -85,B 0,C 180,E1 -2781.138,E2 -2781.138} C_VEL
LIN {X 0,Y 687.947,Z 1038.625,A -85,B 0,C 180,E1 -2782.987,E2 -2782.987} C_VEL
LIN {X 0,Y 687.915,Z 1043.411,A -85,B 0,C 180,E1 -2784.997,E2 -2784.997} C_VEL
LIN {X 0,Y 687.909,Z 1046.288,A -85,B 0,C 180,E1 -2786.75,E2 -2786.75} C_VEL
LIN {X 0,Y 687.91,Z 1048.181,A -85,B 0,C 180,E1 -2788.834,E2 -2788.834} C_VEL
LIN {X 0,Y 687.895,Z 1048.34,A -85,B 0,C 180,E1 -2790.666,E2 -2790.666} C_VEL
LIN {X 0,Y 687.903,Z 1047.264,A -85,B 0,C 180,E1 -2792.499,E2 -2792.499} C_VEL
LIN {X 0,Y 687.917,Z 1044.376,A -85,B 0,C 180,E1 -2794.585,E2 -2794.585} C_VEL
LIN {X 0,Y 687.922,Z 1040.594,A -85,B 0,C 180,E1 -2796.342,E2 -2796.342} C_VEL
LIN {X 0,Y 687.968,Z 1034.797,A -85,B 0,C 180,E1 -2798.357,E2 -2798.357} C_VEL
LIN {X 0,Y 688.05,Z 1027.361,A -85,B 0,C 180,E1 -2800.315,E2 -2800.315} C_VEL
LIN {X 0,Y 688.183,Z 1018.515,A -85,B 0,C 180,E1 -2802.247,E2 -2802.247} C_VEL
LIN {X 0,Y 688.39,Z 1007.592,A -85,B 0,C 180,E1 -2804.21,E2 -2804.21} C_VEL
LIN {X 0,Y 688.675,Z 995.904,A -85,B 0,C 180,E1 -2806.02,E2 -2806.02} C_VEL
LIN {X 0,Y 689.058,Z 982.22,A -85,B 0,C 180,E1 -2807.838,E2 -2807.838} C_VEL
LIN {X 0,Y 689.529,Z 967.366,A -85,B 0,C 180,E1 -2809.571,E2 -2809.571} C_VEL
LIN {X 0,Y 690.129,Z 950.929,A -85,B 0,C 180,E1 -2811.236,E2 -2811.236} C_VEL
LIN {X 0,Y 690.814,Z 933.25,A -85,B 0,C 180,E1 -2812.824,E2 -2812.824} C_VEL
LIN {X 0,Y 691.568,Z 914.44,A -85,B 0,C 180,E1 -2814.289,E2 -2814.289} C_VEL
LIN {X 0,Y 692.399,Z 894.344,A -85,B 0,C 180,E1 -2815.673,E2 -2815.673} C_VEL
LIN {X 0,Y 693.228,Z 873.924,A -85,B 0,C 180,E1 -2816.884,E2 -2816.884} C_VEL
LIN {X 0,Y 694.091,Z 852.204,A -85,B 0,C 180,E1 -2818.01,E2 -2818.01} C_VEL
LIN {X 0,Y 694.881,Z 830.216,A -85,B 0,C 180,E1 -2818.969,E2 -2818.969} C_VEL
LIN {X 0,Y 695.613,Z 809.262,A -85,B 0,C 180,E1 -2819.749,E2 -2819.749} C_VEL
LIN {X 0,Y 696.279,Z 784.512,A -85,B 0,C 180,E1 -2820.5,E2 -2820.5} C_VEL
LIN {X 0,Y 696.849,Z 762.706,A -85,B 0,C 180,E1 -2821.019,E2 -2821.019} C_VEL
LIN {X 0,Y 697.351,Z 737.268,A -85,B 0,C 180,E1 -2821.464,E2 -2821.464} C_VEL
LIN {X 0,Y 698.396,Z 597.859,A -85,B 0,C 180,E1 -2823.098,E2 -2823.098} C_VEL
LIN {X 0,Y 700.129,Z 364.063,A -85,B 0,C 180,E1 -2825.852,E2 -2825.852} C_VEL
LIN {X 0,Y 697.963,Z 356.931,A -85,B 0,C 180,E1 -2826.069,E2 -2826.069} C_VEL
LIN {X 0,Y 692.574,Z 347.312,A -85,B 0,C 180,E1 -2826.54,E2 -2826.54} C_VEL
LIN {X 0,Y 688.439,Z 335.47,A -85,B 0,C 180,E1 -2827.804,E2 -2827.804} C_VEL
LIN {X 0,Y 688.397,Z 335.48,A -85,B 0,C 180,E1 -2830.566,E2 -2830.566} C_VEL
LIN {X 0,Y 688.463,Z 335.458,A -85,B 0,C 180,E1 -2833.433,E2 -2833.433} C_VEL
LIN {X 0,Y 688.401,Z 335.477,A -85,B 0,C 180,E1 -2836.375,E2 -2836.375} C_VEL
LIN {X 0,Y 688.415,Z 335.459,A -85,B 0,C 180,E1 -2839.076,E2 -2839.076} C_VEL
LIN {X 0,Y 688.42,Z 335.47,A -85,B 0,C 180,E1 -2842.198,E2 -2842.198} C_VEL
LIN {X 0,Y 688.398,Z 335.476,A -85,B 0,C 180,E1 -2844.887,E2 -2844.887} C_VEL
LIN {X 0,Y 688.468,Z 335.471,A -85,B 0,C 180,E1 -2847.791,E2 -2847.791} C_VEL
LIN {X 0,Y 688.398,Z 335.475,A -85,B 0,C 180,E1 -2850.693,E2 -2850.693} C_VEL
LIN {X 0,Y 688.417,Z 335.472,A -85,B 0,C 180,E1 -2853.333,E2 -2853.333} C_VEL
LIN {X 0,Y 688.418,Z 335.468,A -85,B 0,C 180,E1 -2856.458,E2 -2856.458} C_VEL
LIN {X 0,Y 688.395,Z 335.475,A -85,B 0,C 180,E1 -2859.065,E2 -2859.065} C_VEL
LIN {X 0,Y 688.466,Z 335.476,A -85,B 0,C 180,E1 -2861.892,E2 -2861.892} C_VEL
LIN {X 0,Y 688.398,Z 335.468,A -85,B 0,C 180,E1 -2864.844,E2 -2864.844} C_VEL
LIN {X 0,Y 688.411,Z 335.477,A -85,B 0,C 180,E1 -2867.501,E2 -2867.501} C_VEL
LIN {X 0,Y 688.424,Z 335.472,A -85,B 0,C 180,E1 -2870.638,E2 -2870.638} C_VEL
LIN {X 0,Y 688.395,Z 335.472,A -85,B 0,C 180,E1 -2873.327,E2 -2873.327} C_VEL
LIN {X 0,Y 688.467,Z 335.473,A -85,B 0,C 180,E1 -2876.253,E2 -2876.253} C_VEL
LIN {X 0,Y 688.395,Z 335.47,A -85,B 0,C 180,E1 -2879.168,E2 -2879.168} C_VEL
LIN {X 0,Y 688.418,Z 335.477,A -85,B 0,C 180,E1 -2881.831,E2 -2881.831} C_VEL
LIN {X 0,Y 688.41,Z 335.473,A -85,B 0,C 180,E1 -2885,E2 -2885} C_VEL
LIN {X 0,Y 688.395,Z 335.471,A -85,B 0,C 180,E1 -2887.595,E2 -2887.595} C_VEL
LIN {X 0,Y 688.466,Z 335.471,A -85,B 0,C 180,E1 -2890.544,E2 -2890.544} C_VEL
LIN {X 0,Y 688.394,Z 335.472,A -85,B 0,C 180,E1 -2893.438,E2 -2893.438} C_VEL
LIN {X 0,Y 688.422,Z 335.476,A -85,B 0,C 180,E1 -2896.106,E2 -2896.106} C_VEL
LIN {X 0,Y 688.408,Z 335.472,A -85,B 0,C 180,E1 -2899.251,E2 -2899.251} C_VEL
LIN {X 0,Y 688.399,Z 335.473,A -85,B 0,C 180,E1 -2901.919,E2 -2901.919} C_VEL
LIN {X 0,Y 688.461,Z 335.471,A -85,B 0,C 180,E1 -2904.909,E2 -2904.909} C_VEL
LIN {X 0,Y 688.394,Z 335.472,A -85,B 0,C 180,E1 -2907.697,E2 -2907.697} C_VEL
LIN {X 0,Y 688.425,Z 335.479,A -85,B 0,C 180,E1 -2910.374,E2 -2910.374} C_VEL
LIN {X 0,Y 688.409,Z 335.473,A -85,B 0,C 180,E1 -2913.5,E2 -2913.5} C_VEL
LIN {X 0,Y 688.397,Z 335.478,A -85,B 0,C 180,E1 -2916.139,E2 -2916.139} C_VEL
LIN {X 0,Y 688.467,Z 335.468,A -85,B 0,C 180,E1 -2919.074,E2 -2919.074} C_VEL
LIN {X 0,Y 688.393,Z 335.471,A -85,B 0,C 180,E1 -2921.954,E2 -2921.954} C_VEL
LIN {X 0,Y 688.432,Z 335.476,A -85,B 0,C 180,E1 -2924.666,E2 -2924.666} C_VEL
LIN {X 0,Y 688.409,Z 335.475,A -85,B 0,C 180,E1 -2927.74,E2 -2927.74} C_VEL
LIN {X 0,Y 688.407,Z 335.581,A -85,B 0,C 180,E1 -2930.113,E2 -2930.113} C_VEL
LIN {X 0,Y 696.631,Z 357.316,A -85,B 0,C 180,E1 -2932.306,E2 -2932.306} C_VEL
LIN {X 0,Y 696.264,Z 377.415,A -85,B 0,C 180,E1 -2933.755,E2 -2933.755} C_VEL
LIN {X 0,Y 700.173,Z 394.081,A -85,B 0,C 180,E1 -2934.196,E2 -2934.196} C_VEL
LIN {X 0,Y 698.2,Z 655.079,A -85,B 0,C 180,E1 -2937.264,E2 -2937.264} C_VEL
LIN {X 0,Y 697.347,Z 767.395,A -85,B 0,C 180,E1 -2938.583,E2 -2938.583} C_VEL
LIN {X 0,Y 696.839,Z 792.887,A -85,B 0,C 180,E1 -2939.03,E2 -2939.03} C_VEL
LIN {X 0,Y 696.274,Z 814.667,A -85,B 0,C 180,E1 -2939.549,E2 -2939.549} C_VEL
LIN {X 0,Y 695.638,Z 838.555,A -85,B 0,C 180,E1 -2940.271,E2 -2940.271} C_VEL
LIN {X 0,Y 694.912,Z 859.351,A -85,B 0,C 180,E1 -2941.041,E2 -2941.041} C_VEL
LIN {X 0,Y 694.116,Z 881.25,A -85,B 0,C 180,E1 -2941.991,E2 -2941.991} C_VEL
LIN {X 0,Y 693.259,Z 903.135,A -85,B 0,C 180,E1 -2943.117,E2 -2943.117} C_VEL
LIN {X 0,Y 692.485,Z 922.178,A -85,B 0,C 180,E1 -2944.239,E2 -2944.239} C_VEL
LIN {X 0,Y 691.611,Z 943.229,A -85,B 0,C 180,E1 -2945.667,E2 -2945.667} C_VEL
LIN {X 0,Y 690.895,Z 961.055,A -85,B 0,C 180,E1 -2947.044,E2 -2947.044} C_VEL
LIN {X 0,Y 690.21,Z 978.604,A -85,B 0,C 180,E1 -2948.588,E2 -2948.588} C_VEL
LIN {X 0,Y 689.672,Z 993.637,A -85,B 0,C 180,E1 -2950.08,E2 -2950.08} C_VEL
LIN {X 0,Y 689.135,Z 1009.812,A -85,B 0,C 180,E1 -2951.911,E2 -2951.911} C_VEL
LIN {X 0,Y 688.749,Z 1022.529,A -85,B 0,C 180,E1 -2953.555,E2 -2953.555} C_VEL
LIN {X 0,Y 688.429,Z 1035.761,A -85,B 0,C 180,E1 -2955.533,E2 -2955.533} C_VEL
LIN {X 0,Y 688.23,Z 1045.568,A -85,B 0,C 180,E1 -2957.242,E2 -2957.242} C_VEL
LIN {X 0,Y 688.07,Z 1055.475,A -85,B 0,C 180,E1 -2959.28,E2 -2959.28} C_VEL
LIN {X 0,Y 687.974,Z 1062.513,A -85,B 0,C 180,E1 -2961.053,E2 -2961.053} C_VEL
LIN {X 0,Y 687.953,Z 1068.506,A -85,B 0,C 180,E1 -2962.903,E2 -2962.903} C_VEL
LIN {X 0,Y 687.923,Z 1073.497,A -85,B 0,C 180,E1 -2964.997,E2 -2964.997} C_VEL
LIN {X 0,Y 687.916,Z 1076.461,A -85,B 0,C 180,E1 -2966.834,E2 -2966.834} C_VEL
LIN {X 0,Y 687.914,Z 1078.239,A -85,B 0,C 180,E1 -2969.001,E2 -2969.001} C_VEL
LIN {X 0,Y 687.898,Z 1078.306,A -85,B 0,C 180,E1 -2970.749,E2 -2970.749} C_VEL
LIN {X 0,Y 687.907,Z 1077.017,A -85,B 0,C 180,E1 -2972.749,E2 -2972.749} C_VEL
LIN {X 0,Y 687.92,Z 1073.973,A -85,B 0,C 180,E1 -2974.752,E2 -2974.752} C_VEL
LIN {X 0,Y 687.916,Z 1070.07,A -85,B 0,C 180,E1 -2976.51,E2 -2976.51} C_VEL
LIN {X 0,Y 687.961,Z 1063.726,A -85,B 0,C 180,E1 -2978.61,E2 -2978.61} C_VEL
LIN {X 0,Y 688.057,Z 1056.895,A -85,B 0,C 180,E1 -2980.381,E2 -2980.381} C_VEL
LIN {X 0,Y 688.19,Z 1047.864,A -85,B 0,C 180,E1 -2982.332,E2 -2982.332} C_VEL
LIN {X 0,Y 688.386,Z 1037.323,A -85,B 0,C 180,E1 -2984.21,E2 -2984.21} C_VEL
LIN {X 0,Y 688.696,Z 1025.064,A -85,B 0,C 180,E1 -2986.099,E2 -2986.099} C_VEL
LIN {X 0,Y 689.094,Z 1011.228,A -85,B 0,C 180,E1 -2987.916,E2 -2987.916} C_VEL
LIN {X 0,Y 689.579,Z 996.174,A -85,B 0,C 180,E1 -2989.658,E2 -2989.658} C_VEL
LIN {X 0,Y 690.14,Z 980.463,A -85,B 0,C 180,E1 -2991.236,E2 -2991.236} C_VEL
LIN {X 0,Y 690.837,Z 962.714,A -85,B 0,C 180,E1 -2992.823,E2 -2992.823} C_VEL
LIN {X 0,Y 691.588,Z 943.838,A -85,B 0,C 180,E1 -2994.288,E2 -2994.288} C_VEL
LIN {X 0,Y 692.427,Z 923.629,A -85,B 0,C 180,E1 -2995.671,E2 -2995.671} C_VEL
LIN {X 0,Y 693.227,Z 903.945,A -85,B 0,C 180,E1 -2996.837,E2 -2996.837} C_VEL
LIN {X 0,Y 694.091,Z 882.149,A -85,B 0,C 180,E1 -2997.968,E2 -2997.968} C_VEL
LIN {X 0,Y 694.872,Z 860.49,A -85,B 0,C 180,E1 -2998.913,E2 -2998.913} C_VEL
LIN {X 0,Y 695.586,Z 839.844,A -85,B 0,C 180,E1 -2999.684,E2 -2999.684} C_VEL
LIN {X 0,Y 696.271,Z 814.783,A -85,B 0,C 180,E1 -3000.448,E2 -3000.448} C_VEL
LIN {X 0,Y 696.835,Z 793.027,A -85,B 0,C 180,E1 -3000.967,E2 -3000.967} C_VEL
LIN {X 0,Y 697.348,Z 767.548,A -85,B 0,C 180,E1 -3001.415,E2 -3001.415} C_VEL
LIN {X 0,Y 698.176,Z 658.274,A -85,B 0,C 180,E1 -3002.699,E2 -3002.699} C_VEL
LIN {X 0,Y 700.159,Z 395.86,A -85,B 0,C 180,E1 -3005.783,E2 -3005.783} C_VEL
LIN {X 0,Y 699.898,Z 392.055,A -85,B 0,C 180,E1 -3005.846,E2 -3005.846} C_VEL
LIN {X 0,Y 696.185,Z 376.671,A -85,B 0,C 180,E1 -3006.28,E2 -3006.28} C_VEL
LIN {X 0,Y 696.514,Z 357.054,A -85,B 0,C 180,E1 -3007.721,E2 -3007.721} C_VEL
LIN {X 0,Y 689.277,Z 338.254,A -85,B 0,C 180,E1 -3009.62,E2 -3009.62} C_VEL
LIN {X 0,Y 688.394,Z 335.483,A -85,B 0,C 180,E1 -3009.922,E2 -3009.922} C_VEL
LIN {X 0,Y 688.458,Z 335.472,A -85,B 0,C 180,E1 -3012.707,E2 -3012.707} C_VEL
LIN {X 0,Y 688.401,Z 335.477,A -85,B 0,C 180,E1 -3015.681,E2 -3015.681} C_VEL
LIN {X 0,Y 688.404,Z 335.473,A -85,B 0,C 180,E1 -3018.299,E2 -3018.299} C_VEL
LIN {X 0,Y 688.445,Z 335.478,A -85,B 0,C 180,E1 -3021.352,E2 -3021.352} C_VEL
LIN {X 0,Y 688.393,Z 335.453,A -85,B 0,C 180,E1 -3024.144,E2 -3024.144} C_VEL
LIN {X 0,Y 688.464,Z 335.468,A -85,B 0,C 180,E1 -3027,E2 -3027} C_VEL
LIN {X 0,Y 688.401,Z 335.475,A -85,B 0,C 180,E1 -3029.96,E2 -3029.96} C_VEL
LIN {X 0,Y 688.408,Z 335.467,A -85,B 0,C 180,E1 -3032.585,E2 -3032.585} C_VEL
LIN {X 0,Y 688.44,Z 335.472,A -85,B 0,C 180,E1 -3035.639,E2 -3035.639} C_VEL
LIN {X 0,Y 688.396,Z 335.474,A -85,B 0,C 180,E1 -3038.371,E2 -3038.371} C_VEL
LIN {X 0,Y 688.466,Z 335.469,A -85,B 0,C 180,E1 -3041.249,E2 -3041.249} C_VEL
LIN {X 0,Y 688.4,Z 335.472,A -85,B 0,C 180,E1 -3044.24,E2 -3044.24} C_VEL
LIN {X 0,Y 688.415,Z 335.472,A -85,B 0,C 180,E1 -3046.904,E2 -3046.904} C_VEL
LIN {X 0,Y 688.421,Z 335.477,A -85,B 0,C 180,E1 -3050.047,E2 -3050.047} C_VEL
LIN {X 0,Y 688.398,Z 335.466,A -85,B 0,C 180,E1 -3052.74,E2 -3052.74} C_VEL
LIN {X 0,Y 688.467,Z 335.475,A -85,B 0,C 180,E1 -3055.669,E2 -3055.669} C_VEL
LIN {X 0,Y 688.399,Z 335.474,A -85,B 0,C 180,E1 -3058.585,E2 -3058.585} C_VEL
LIN {X 0,Y 688.438,Z 335.469,A -85,B 0,C 180,E1 -3061.332,E2 -3061.332} C_VEL
LIN {X 0,Y 688.412,Z 335.476,A -85,B 0,C 180,E1 -3064.415,E2 -3064.415} C_VEL
LIN {X 0,Y 688.405,Z 335.466,A -85,B 0,C 180,E1 -3067.092,E2 -3067.092} C_VEL
LIN {X 0,Y 688.456,Z 335.473,A -85,B 0,C 180,E1 -3070.122,E2 -3070.122} C_VEL
LIN {X 0,Y 688.399,Z 335.474,A -85,B 0,C 180,E1 -3072.937,E2 -3072.937} C_VEL
LIN {X 0,Y 688.462,Z 335.467,A -85,B 0,C 180,E1 -3075.759,E2 -3075.759} C_VEL
LIN {X 0,Y 688.408,Z 335.474,A -85,B 0,C 180,E1 -3078.736,E2 -3078.736} C_VEL
LIN {X 0,Y 688.413,Z 335.471,A -85,B 0,C 180,E1 -3081.405,E2 -3081.405} C_VEL
LIN {X 0,Y 688.448,Z 335.473,A -85,B 0,C 180,E1 -3084.452,E2 -3084.452} C_VEL
LIN {X 0,Y 688.402,Z 335.471,A -85,B 0,C 180,E1 -3087.263,E2 -3087.263} C_VEL
LIN {X 0,Y 688.416,Z 335.469,A -85,B 0,C 180,E1 -3087.56,E2 -3087.56} C_VEL
LIN {X 0,Y 687.48,Z 335.592,A -85,B 0,C 180,E1 -3088.2,E2 -3088.2} C_VEL
LIN {X 0,Y 681.004,Z 336.409,A -85,B 0,C 180,E1 -3090.043,E2 -3090.043} C_VEL
LIN {X 0,Y 680.522,Z 336.461,A -85,B 0,C 180,E1 -3090.464,E2 -3090.464} C_VEL
LIN {X 0,Y 680.463,Z 336.463,A -85,B 0,C 180,E1 -3093.337,E2 -3093.337} C_VEL
LIN {X 0,Y 680.528,Z 336.46,A -85,B 0,C 180,E1 -3096.231,E2 -3096.231} C_VEL
LIN {X 0,Y 680.467,Z 336.465,A -85,B 0,C 180,E1 -3099.187,E2 -3099.187} C_VEL
LIN {X 0,Y 680.496,Z 336.462,A -85,B 0,C 180,E1 -3101.97,E2 -3101.97} C_VEL
LIN {X 0,Y 680.479,Z 336.465,A -85,B 0,C 180,E1 -3105.093,E2 -3105.093} C_VEL
LIN {X 0,Y 680.473,Z 336.465,A -85,B 0,C 180,E1 -3107.816,E2 -3107.816} C_VEL
LIN {X 0,Y 680.514,Z 336.467,A -85,B 0,C 180,E1 -3110.878,E2 -3110.878} C_VEL
LIN {X 0,Y 680.488,Z 336.593,A -85,B 0,C 180,E1 -3111.845,E2 -3111.845} C_VEL
LIN {X 0,Y 684.757,Z 348.307,A -85,B 0,C 180,E1 -3113.097,E2 -3113.097} C_VEL
LIN {X 0,Y 692.725,Z 362.511,A -85,B 0,C 180,E1 -3113.774,E2 -3113.774} C_VEL
LIN {X 0,Y 693.619,Z 366.828,A -85,B 0,C 180,E1 -3113.883,E2 -3113.883} C_VEL
LIN {X 0,Y 691.621,Z 606.508,A -85,B 0,C 180,E1 -3116.732,E2 -3116.732} C_VEL
LIN {X 0,Y 690.513,Z 737.342,A -85,B 0,C 180,E1 -3118.28,E2 -3118.28} C_VEL
LIN {X 0,Y 689.958,Z 762.788,A -85,B 0,C 180,E1 -3118.729,E2 -3118.729} C_VEL
LIN {X 0,Y 689.331,Z 784.468,A -85,B 0,C 180,E1 -3119.249,E2 -3119.249} C_VEL
LIN {X 0,Y 688.601,Z 808.637,A -85,B 0,C 180,E1 -3119.985,E2 -3119.985} C_VEL
LIN {X 0,Y 687.8,Z 829.42,A -85,B 0,C 180,E1 -3120.761,E2 -3120.761} C_VEL
LIN {X 0,Y 686.914,Z 851.384,A -85,B 0,C 180,E1 -3121.722,E2 -3121.722} C_VEL
LIN {X 0,Y 685.945,Z 873.163,A -85,B 0,C 180,E1 -3122.854,E2 -3122.854} C_VEL
LIN {X 0,Y 685.052,Z 893.075,A -85,B 0,C 180,E1 -3124.041,E2 -3124.041} C_VEL
LIN {X 0,Y 684.092,Z 913.24,A -85,B 0,C 180,E1 -3125.428,E2 -3125.428} C_VEL
LIN {X 0,Y 683.302,Z 931.065,A -85,B 0,C 180,E1 -3126.819,E2 -3126.819} C_VEL
LIN {X 0,Y 682.506,Z 949.073,A -85,B 0,C 180,E1 -3128.425,E2 -3128.425} C_VEL
LIN {X 0,Y 681.86,Z 965.153,A -85,B 0,C 180,E1 -3130.048,E2 -3130.048} C_VEL
LIN {X 0,Y 681.267,Z 980.87,A -85,B 0,C 180,E1 -3131.871,E2 -3131.871} C_VEL
LIN {X 0,Y 680.814,Z 994.744,A -85,B 0,C 180,E1 -3133.709,E2 -3133.709} C_VEL
LIN {X 0,Y 680.473,Z 1007.056,A -85,B 0,C 180,E1 -3135.621,E2 -3135.621} C_VEL
LIN {X 0,Y 680.242,Z 1017.623,A -85,B 0,C 180,E1 -3137.521,E2 -3137.521} C_VEL
LIN {X 0,Y 680.077,Z 1026.709,A -85,B 0,C 180,E1 -3139.496,E2 -3139.496} C_VEL
LIN {X 0,Y 679.969,Z 1033.566,A -85,B 0,C 180,E1 -3141.288,E2 -3141.288} C_VEL
LIN {X 0,Y 679.93,Z 1039.961,A -85,B 0,C 180,E1 -3143.413,E2 -3143.413} C_VEL
LIN {X 0,Y 679.91,Z 1043.889,A -85,B 0,C 180,E1 -3145.192,E2 -3145.192} C_VEL
LIN {X 0,Y 679.903,Z 1046.851,A -85,B 0,C 180,E1 -3147.134,E2 -3147.134} C_VEL
LIN {X 0,Y 679.903,Z 1048.272,A -85,B 0,C 180,E1 -3149.157,E2 -3149.157} C_VEL
LIN {X 0,Y 679.909,Z 1048.273,A -85,B 0,C 180,E1 -3150.927,E2 -3150.927} C_VEL
LIN {X 0,Y 679.91,Z 1046.689,A -85,B 0,C 180,E1 -3153.078,E2 -3153.078} C_VEL
LIN {X 0,Y 679.915,Z 1043.899,A -85,B 0,C 180,E1 -3154.893,E2 -3154.893} C_VEL
LIN {X 0,Y 679.931,Z 1039.767,A -85,B 0,C 180,E1 -3156.756,E2 -3156.756} C_VEL
LIN {X 0,Y 679.971,Z 1033.5,A -85,B 0,C 180,E1 -3158.82,E2 -3158.82} C_VEL
LIN {X 0,Y 680.079,Z 1026.727,A -85,B 0,C 180,E1 -3160.59,E2 -3160.59} C_VEL
LIN {X 0,Y 680.243,Z 1017.6,A -85,B 0,C 180,E1 -3162.573,E2 -3162.573} C_VEL
LIN {X 0,Y 680.475,Z 1007.07,A -85,B 0,C 180,E1 -3164.466,E2 -3164.466} C_VEL
LIN {X 0,Y 680.817,Z 994.757,A -85,B 0,C 180,E1 -3166.379,E2 -3166.379} C_VEL
LIN {X 0,Y 681.267,Z 980.881,A -85,B 0,C 180,E1 -3168.217,E2 -3168.217} C_VEL
LIN {X 0,Y 681.835,Z 965.751,A -85,B 0,C 180,E1 -3169.98,E2 -3169.98} C_VEL
LIN {X 0,Y 682.468,Z 949.995,A -85,B 0,C 180,E1 -3171.577,E2 -3171.577} C_VEL
LIN {X 0,Y 683.256,Z 932.153,A -85,B 0,C 180,E1 -3173.182,E2 -3173.182} C_VEL
LIN {X 0,Y 684.071,Z 913.821,A -85,B 0,C 180,E1 -3174.619,E2 -3174.619} C_VEL
LIN {X 0,Y 685.027,Z 893.75,A -85,B 0,C 180,E1 -3176.007,E2 -3176.007} C_VEL
LIN {X 0,Y 685.919,Z 873.828,A -85,B 0,C 180,E1 -3177.199,E2 -3177.199} C_VEL
LIN {X 0,Y 686.885,Z 852.193,A -85,B 0,C 180,E1 -3178.33,E2 -3178.33} C_VEL
LIN {X 0,Y 687.76,Z 830.415,A -85,B 0,C 180,E1 -3179.289,E2 -3179.289} C_VEL
LIN {X 0,Y 688.512,Z 810.911,A -85,B 0,C 180,E1 -3180.025,E2 -3180.025} C_VEL
LIN {X 0,Y 689.307,Z 785.494,A -85,B 0,C 180,E1 -3180.813,E2 -3180.813} C_VEL
LIN {X 0,Y 689.924,Z 763.903,A -85,B 0,C 180,E1 -3181.337,E2 -3181.337} C_VEL
LIN {X 0,Y 690.507,Z 738.165,A -85,B 0,C 180,E1 -3181.799,E2 -3181.799} C_VEL
LIN {X 0,Y 691.217,Z 657.187,A -85,B 0,C 180,E1 -3182.765,E2 -3182.765} C_VEL
LIN {X 0,Y 693.246,Z 409.554,A -85,B 0,C 180,E1 -3185.694,E2 -3185.694} C_VEL
LIN {X 0,Y 693.447,Z 365.242,A -85,B 0,C 180,E1 -3186.237,E2 -3186.237} C_VEL
LIN {X 0,Y 692.045,Z 361.023,A -85,B 0,C 180,E1 -3186.376,E2 -3186.376} C_VEL
LIN {X 0,Y 684.473,Z 347.75,A -85,B 0,C 180,E1 -3187.028,E2 -3187.028} C_VEL
LIN {X 0,Y 680.461,Z 336.471,A -85,B 0,C 180,E1 -3188.27,E2 -3188.27} C_VEL
LIN {X 0,Y 680.479,Z 336.466,A -85,B 0,C 180,E1 -3190.951,E2 -3190.951} C_VEL
LIN {X 0,Y 680.472,Z 336.449,A -85,B 0,C 180,E1 -3194.147,E2 -3194.147} C_VEL
LIN {X 0,Y 680.461,Z 336.468,A -85,B 0,C 180,E1 -3196.789,E2 -3196.789} C_VEL
LIN {X 0,Y 680.524,Z 336.455,A -85,B 0,C 180,E1 -3199.821,E2 -3199.821} C_VEL
LIN {X 0,Y 680.456,Z 336.461,A -85,B 0,C 180,E1 -3202.652,E2 -3202.652} C_VEL
LIN {X 0,Y 680.507,Z 336.463,A -85,B 0,C 180,E1 -3205.447,E2 -3205.447} C_VEL
LIN {X 0,Y 680.468,Z 336.459,A -85,B 0,C 180,E1 -3208.459,E2 -3208.459} C_VEL
LIN {X 0,Y 680.462,Z 336.466,A -85,B 0,C 180,E1 -3211.089,E2 -3211.089} C_VEL
LIN {X 0,Y 680.523,Z 336.461,A -85,B 0,C 180,E1 -3214.055,E2 -3214.055} C_VEL
LIN {X 0,Y 680.455,Z 336.459,A -85,B 0,C 180,E1 -3216.907,E2 -3216.907} C_VEL
LIN {X 0,Y 680.511,Z 336.462,A -85,B 0,C 180,E1 -3219.711,E2 -3219.711} C_VEL
LIN {X 0,Y 680.463,Z 336.463,A -85,B 0,C 180,E1 -3222.771,E2 -3222.771} C_VEL
LIN {X 0,Y 680.469,Z 336.459,A -85,B 0,C 180,E1 -3225.447,E2 -3225.447} C_VEL
LIN {X 0,Y 680.488,Z 336.454,A -85,B 0,C 180,E1 -3228.559,E2 -3228.559} C_VEL
LIN {X 0,Y 680.457,Z 336.464,A -85,B 0,C 180,E1 -3231.295,E2 -3231.295} C_VEL
LIN {X 0,Y 680.529,Z 336.458,A -85,B 0,C 180,E1 -3234.181,E2 -3234.181} C_VEL
LIN {X 0,Y 680.456,Z 336.462,A -85,B 0,C 180,E1 -3237.136,E2 -3237.136} C_VEL
LIN {X 0,Y 680.483,Z 336.462,A -85,B 0,C 180,E1 -3239.832,E2 -3239.832} C_VEL
LIN {X 0,Y 680.473,Z 336.453,A -85,B 0,C 180,E1 -3242.948,E2 -3242.948} C_VEL
LIN {X 0,Y 680.461,Z 336.465,A -85,B 0,C 180,E1 -3245.65,E2 -3245.65} C_VEL
LIN {X 0,Y 680.523,Z 336.46,A -85,B 0,C 180,E1 -3248.619,E2 -3248.619} C_VEL
LIN {X 0,Y 680.455,Z 336.461,A -85,B 0,C 180,E1 -3251.444,E2 -3251.444} C_VEL
LIN {X 0,Y 680.5,Z 336.465,A -85,B 0,C 180,E1 -3254.204,E2 -3254.204} C_VEL
LIN {X 0,Y 680.466,Z 336.459,A -85,B 0,C 180,E1 -3257.267,E2 -3257.267} C_VEL
LIN {X 0,Y 680.463,Z 336.464,A -85,B 0,C 180,E1 -3259.932,E2 -3259.932} C_VEL
LIN {X 0,Y 680.52,Z 336.459,A -85,B 0,C 180,E1 -3262.915,E2 -3262.915} C_VEL
LIN {X 0,Y 680.455,Z 336.463,A -85,B 0,C 180,E1 -3265.741,E2 -3265.741} C_VEL
LIN {X 0,Y 680.523,Z 336.46,A -85,B 0,C 180,E1 -3268.62,E2 -3268.62} C_VEL
LIN {X 0,Y 680.463,Z 336.46,A -85,B 0,C 180,E1 -3271.542,E2 -3271.542} C_VEL
LIN {X 0,Y 680.464,Z 336.465,A -85,B 0,C 180,E1 -3274.179,E2 -3274.179} C_VEL
LIN {X 0,Y 680.505,Z 336.461,A -85,B 0,C 180,E1 -3277.255,E2 -3277.255} C_VEL
LIN {X 0,Y 680.454,Z 336.459,A -85,B 0,C 180,E1 -3280.041,E2 -3280.041} C_VEL
LIN {X 0,Y 680.519,Z 336.465,A -85,B 0,C 180,E1 -3282.866,E2 -3282.866} C_VEL
LIN {X 0,Y 680.46,Z 336.463,A -85,B 0,C 180,E1 -3285.852,E2 -3285.852} C_VEL
LIN {X 0,Y 680.472,Z 336.469,A -85,B 0,C 180,E1 -3288.539,E2 -3288.539} C_VEL
LIN {X 0,Y 680.492,Z 336.544,A -85,B 0,C 180,E1 -3289.651,E2 -3289.651} C_VEL
LIN {X 0,Y 689.626,Z 360.88,A -85,B 0,C 180,E1 -3292.143,E2 -3292.143} C_VEL
LIN {X 0,Y 689.265,Z 377.17,A -85,B 0,C 180,E1 -3293.327,E2 -3293.327} C_VEL
LIN {X 0,Y 693.662,Z 395.742,A -85,B 0,C 180,E1 -3293.828,E2 -3293.828} C_VEL
LIN {X 0,Y 691.448,Z 657.37,A -85,B 0,C 180,E1 -3296.931,E2 -3296.931} C_VEL
LIN {X 0,Y 690.51,Z 767.572,A -85,B 0,C 180,E1 -3298.238,E2 -3298.238} C_VEL
LIN {X 0,Y 689.947,Z 793.145,A -85,B 0,C 180,E1 -3298.692,E2 -3298.692} C_VEL
LIN {X 0,Y 689.322,Z 814.773,A -85,B 0,C 180,E1 -3299.212,E2 -3299.212} C_VEL
LIN {X 0,Y 688.555,Z 839.836,A -85,B 0,C 180,E1 -3299.982,E2 -3299.982} C_VEL
LIN {X 0,Y 687.759,Z 860.479,A -85,B 0,C 180,E1 -3300.759,E2 -3300.759} C_VEL
LIN {X 0,Y 686.833,Z 883.157,A -85,B 0,C 180,E1 -3301.762,E2 -3301.762} C_VEL
LIN {X 0,Y 685.914,Z 903.943,A -85,B 0,C 180,E1 -3302.853,E2 -3302.853} C_VEL
LIN {X 0,Y 685,Z 924.289,A -85,B 0,C 180,E1 -3304.071,E2 -3304.071} C_VEL
LIN {X 0,Y 684.046,Z 944.443,A -85,B 0,C 180,E1 -3305.472,E2 -3305.472} C_VEL
LIN {X 0,Y 683.213,Z 963.249,A -85,B 0,C 180,E1 -3306.953,E2 -3306.953} C_VEL
LIN {X 0,Y 682.445,Z 980.46,A -85,B 0,C 180,E1 -3308.513,E2 -3308.513} C_VEL
LIN {X 0,Y 681.781,Z 996.971,A -85,B 0,C 180,E1 -3310.197,E2 -3310.197} C_VEL
LIN {X 0,Y 681.235,Z 1011.929,A -85,B 0,C 180,E1 -3311.959,E2 -3311.959} C_VEL
LIN {X 0,Y 680.769,Z 1026.226,A -85,B 0,C 180,E1 -3313.883,E2 -3313.883} C_VEL
LIN {X 0,Y 680.444,Z 1037.837,A -85,B 0,C 180,E1 -3315.708,E2 -3315.708} C_VEL
LIN {X 0,Y 680.212,Z 1048.708,A -85,B 0,C 180,E1 -3317.693,E2 -3317.693} C_VEL
LIN {X 0,Y 680.072,Z 1057.251,A -85,B 0,C 180,E1 -3319.581,E2 -3319.581} C_VEL
LIN {X 0,Y 679.972,Z 1064.635,A -85,B 0,C 180,E1 -3321.544,E2 -3321.544} C_VEL
LIN {X 0,Y 679.918,Z 1070.277,A -85,B 0,C 180,E1 -3323.498,E2 -3323.498} C_VEL
LIN {X 0,Y 679.92,Z 1074.132,A -85,B 0,C 180,E1 -3325.276,E2 -3325.276} C_VEL
LIN {X 0,Y 679.906,Z 1077.091,A -85,B 0,C 180,E1 -3327.303,E2 -3327.303} C_VEL
LIN {X 0,Y 679.899,Z 1078.306,A -85,B 0,C 180,E1 -3329.242,E2 -3329.242} C_VEL
LIN {X 0,Y 679.914,Z 1078.238,A -85,B 0,C 180,E1 -3331.011,E2 -3331.011} C_VEL
LIN {X 0,Y 679.916,Z 1076.461,A -85,B 0,C 180,E1 -3333.203,E2 -3333.203} C_VEL
LIN {X 0,Y 679.923,Z 1073.497,A -85,B 0,C 180,E1 -3335.062,E2 -3335.062} C_VEL
LIN {X 0,Y 679.954,Z 1068.507,A -85,B 0,C 180,E1 -3337.18,E2 -3337.18} C_VEL
LIN {X 0,Y 679.992,Z 1062.513,A -85,B 0,C 180,E1 -3339.052,E2 -3339.052} C_VEL
LIN {X 0,Y 680.097,Z 1055.12,A -85,B 0,C 180,E1 -3340.933,E2 -3340.933} C_VEL
LIN {X 0,Y 680.283,Z 1045.255,A -85,B 0,C 180,E1 -3342.969,E2 -3342.969} C_VEL
LIN {X 0,Y 680.52,Z 1035.246,A -85,B 0,C 180,E1 -3344.725,E2 -3344.725} C_VEL
LIN {X 0,Y 680.898,Z 1021.894,A -85,B 0,C 180,E1 -3346.728,E2 -3346.728} C_VEL
LIN {X 0,Y 681.318,Z 1009.108,A -85,B 0,C 180,E1 -3348.393,E2 -3348.393} C_VEL
LIN {X 0,Y 681.951,Z 992.792,A -85,B 0,C 180,E1 -3350.244,E2 -3350.244} C_VEL
LIN {X 0,Y 682.561,Z 977.637,A -85,B 0,C 180,E1 -3351.758,E2 -3351.758} C_VEL
LIN {X 0,Y 683.397,Z 958.848,A -85,B 0,C 180,E1 -3353.405,E2 -3353.405} C_VEL
LIN {X 0,Y 684.206,Z 940.793,A -85,B 0,C 180,E1 -3354.798,E2 -3354.798} C_VEL
LIN {X 0,Y 685.183,Z 919.997,A -85,B 0,C 180,E1 -3356.196,E2 -3356.196} C_VEL
LIN {X 0,Y 686.049,Z 900.696,A -85,B 0,C 180,E1 -3357.329,E2 -3357.329} C_VEL
LIN {X 0,Y 687.089,Z 877.283,A -85,B 0,C 180,E1 -3358.511,E2 -3358.511} C_VEL
LIN {X 0,Y 687.891,Z 857.094,A -85,B 0,C 180,E1 -3359.378,E2 -3359.378} C_VEL
LIN {X 0,Y 688.774,Z 832.987,A -85,B 0,C 180,E1 -3360.248,E2 -3360.248} C_VEL
LIN {X 0,Y 689.455,Z 811.01,A -85,B 0,C 180,E1 -3360.886,E2 -3360.886} C_VEL
LIN {X 0,Y 690.144,Z 786.736,A -85,B 0,C 180,E1 -3361.441,E2 -3361.441} C_VEL
LIN {X 0,Y 690.548,Z 763.435,A -85,B 0,C 180,E1 -3361.819,E2 -3361.819} C_VEL
LIN {X 0,Y 692.56,Z 519.708,A -85,B 0,C 180,E1 -3364.693,E2 -3364.693} C_VEL
LIN {X 0,Y 693.501,Z 394.272,A -85,B 0,C 180,E1 -3366.2,E2 -3366.2} C_VEL
LIN {X 0,Y 689.197,Z 376.45,A -85,B 0,C 180,E1 -3366.707,E2 -3366.707} C_VEL
LIN {X 0,Y 689.44,Z 360.313,A -85,B 0,C 180,E1 -3367.911,E2 -3367.911} C_VEL
LIN {X 0,Y 682.411,Z 342.075,A -85,B 0,C 180,E1 -3369.779,E2 -3369.779} C_VEL
LIN {X 0,Y 680.483,Z 336.466,A -85,B 0,C 180,E1 -3370.363,E2 -3370.363} C_VEL
LIN {X 0,Y 680.477,Z 336.466,A -85,B 0,C 180,E1 -3373.457,E2 -3373.457} C_VEL
LIN {X 0,Y 680.457,Z 336.465,A -85,B 0,C 180,E1 -3376.086,E2 -3376.086} C_VEL
LIN {X 0,Y 680.53,Z 336.464,A -85,B 0,C 180,E1 -3379.057,E2 -3379.057} C_VEL
LIN {X 0,Y 680.456,Z 336.464,A -85,B 0,C 180,E1 -3381.964,E2 -3381.964} C_VEL
LIN {X 0,Y 680.502,Z 336.436,A -85,B 0,C 180,E1 -3384.781,E2 -3384.781} C_VEL
LIN {X 0,Y 680.466,Z 336.462,A -85,B 0,C 180,E1 -3387.82,E2 -3387.82} C_VEL
LIN {X 0,Y 680.464,Z 336.461,A -85,B 0,C 180,E1 -3390.447,E2 -3390.447} C_VEL
LIN {X 0,Y 680.517,Z 336.464,A -85,B 0,C 180,E1 -3393.484,E2 -3393.484} C_VEL
LIN {X 0,Y 680.456,Z 336.46,A -85,B 0,C 180,E1 -3396.271,E2 -3396.271} C_VEL
LIN {X 0,Y 680.502,Z 336.46,A -85,B 0,C 180,E1 -3398.991,E2 -3398.991} C_VEL
LIN {X 0,Y 680.472,Z 336.465,A -85,B 0,C 180,E1 -3402.026,E2 -3402.026} C_VEL
LIN {X 0,Y 680.463,Z 336.459,A -85,B 0,C 180,E1 -3404.663,E2 -3404.663} C_VEL
LIN {X 0,Y 680.525,Z 336.46,A -85,B 0,C 180,E1 -3407.613,E2 -3407.613} C_VEL
LIN {X 0,Y 680.458,Z 336.464,A -85,B 0,C 180,E1 -3410.527,E2 -3410.527} C_VEL
LIN {X 0,Y 680.529,Z 336.451,A -85,B 0,C 180,E1 -3413.419,E2 -3413.419} C_VEL
LIN {X 0,Y 680.466,Z 336.46,A -85,B 0,C 180,E1 -3416.377,E2 -3416.377} C_VEL
LIN {X 0,Y 680.474,Z 336.46,A -85,B 0,C 180,E1 -3419.074,E2 -3419.074} C_VEL
LIN {X 0,Y 680.491,Z 336.461,A -85,B 0,C 180,E1 -3422.189,E2 -3422.189} C_VEL
LIN {X 0,Y 680.462,Z 336.462,A -85,B 0,C 180,E1 -3424.95,E2 -3424.95} C_VEL
LIN {X 0,Y 680.528,Z 336.458,A -85,B 0,C 180,E1 -3427.939,E2 -3427.939} C_VEL
LIN {X 0,Y 680.46,Z 336.457,A -85,B 0,C 180,E1 -3430.841,E2 -3430.841} C_VEL
LIN {X 0,Y 680.517,Z 336.459,A -85,B 0,C 180,E1 -3433.684,E2 -3433.684} C_VEL
LIN {X 0,Y 680.474,Z 336.464,A -85,B 0,C 180,E1 -3436.655,E2 -3436.655} C_VEL
LIN {X 0,Y 680.475,Z 336.459,A -85,B 0,C 180,E1 -3439.395,E2 -3439.395} C_VEL
LIN {X 0,Y 680.504,Z 336.465,A -85,B 0,C 180,E1 -3442.459,E2 -3442.459} C_VEL
LIN {X 0,Y 680.462,Z 336.462,A -85,B 0,C 180,E1 -3445.223,E2 -3445.223} C_VEL
LIN {X 0,Y 680.529,Z 336.457,A -85,B 0,C 180,E1 -3448.168,E2 -3448.168} C_VEL
LIN {X 0,Y 680.522,Z 336.461,A -85,B 0,C 180,E1 -3450.464,E2 -3450.464} C_VEL
LIN {X 0,Y 679.468,Z 336.583,A -85,B 0,C 180,E1 -3451.112,E2 -3451.112} C_VEL
LIN {X 0,Y 673.042,Z 337.394,A -85,B 0,C 180,E1 -3452.93,E2 -3452.93} C_VEL
LIN {X 0,Y 672.526,Z 337.452,A -85,B 0,C 180,E1 -3453.403,E2 -3453.403} C_VEL
LIN {X 0,Y 672.589,Z 337.452,A -85,B 0,C 180,E1 -3456.382,E2 -3456.382} C_VEL
LIN {X 0,Y 672.526,Z 337.453,A -85,B 0,C 180,E1 -3459.299,E2 -3459.299} C_VEL
LIN {X 0,Y 672.573,Z 337.451,A -85,B 0,C 180,E1 -3462.111,E2 -3462.111} C_VEL
LIN {X 0,Y 672.533,Z 337.454,A -85,B 0,C 180,E1 -3465.193,E2 -3465.193} C_VEL
LIN {X 0,Y 672.54,Z 337.454,A -85,B 0,C 180,E1 -3467.893,E2 -3467.893} C_VEL
LIN {X 0,Y 672.558,Z 337.458,A -85,B 0,C 180,E1 -3471.036,E2 -3471.036} C_VEL
LIN {X 0,Y 672.558,Z 337.659,A -85,B 0,C 180,E1 -3471.383,E2 -3471.383} C_VEL
LIN {X 0,Y 676.599,Z 348.518,A -85,B 0,C 180,E1 -3472.575,E2 -3472.575} C_VEL
LIN {X 0,Y 686.82,Z 366.468,A -85,B 0,C 180,E1 -3473.46,E2 -3473.46} C_VEL
LIN {X 0,Y 687.145,Z 369.571,A -85,B 0,C 180,E1 -3473.52,E2 -3473.52} C_VEL
LIN {X 0,Y 684.902,Z 609.993,A -85,B 0,C 180,E1 -3476.405,E2 -3476.405} C_VEL
LIN {X 0,Y 683.702,Z 737.492,A -85,B 0,C 180,E1 -3477.928,E2 -3477.928} C_VEL
LIN {X 0,Y 683.096,Z 762.943,A -85,B 0,C 180,E1 -3478.382,E2 -3478.382} C_VEL
LIN {X 0,Y 682.42,Z 784.379,A -85,B 0,C 180,E1 -3478.9,E2 -3478.9} C_VEL
LIN {X 0,Y 681.595,Z 808.649,A -85,B 0,C 180,E1 -3479.644,E2 -3479.644} C_VEL
LIN {X 0,Y 680.714,Z 829.43,A -85,B 0,C 180,E1 -3480.426,E2 -3480.426} C_VEL
LIN {X 0,Y 679.79,Z 850.334,A -85,B 0,C 180,E1 -3481.347,E2 -3481.347} C_VEL
LIN {X 0,Y 678.694,Z 872.263,A -85,B 0,C 180,E1 -3482.487,E2 -3482.487} C_VEL
LIN {X 0,Y 677.745,Z 891.487,A -85,B 0,C 180,E1 -3483.636,E2 -3483.636} C_VEL
LIN {X 0,Y 676.627,Z 912.637,A -85,B 0,C 180,E1 -3485.092,E2 -3485.092} C_VEL
LIN {X 0,Y 675.749,Z 930.521,A -85,B 0,C 180,E1 -3486.499,E2 -3486.499} C_VEL
LIN {X 0,Y 674.826,Z 949.079,A -85,B 0,C 180,E1 -3488.167,E2 -3488.167} C_VEL
LIN {X 0,Y 674.121,Z 964.905,A -85,B 0,C 180,E1 -3489.782,E2 -3489.782} C_VEL
LIN {X 0,Y 673.452,Z 980.263,A -85,B 0,C 180,E1 -3491.576,E2 -3491.576} C_VEL
LIN {X 0,Y 672.977,Z 993.476,A -85,B 0,C 180,E1 -3493.336,E2 -3493.336} C_VEL
LIN {X 0,Y 672.566,Z 1006.541,A -85,B 0,C 180,E1 -3495.361,E2 -3495.361} C_VEL
LIN {X 0,Y 672.308,Z 1016.25,A -85,B 0,C 180,E1 -3497.11,E2 -3497.11} C_VEL
LIN {X 0,Y 672.099,Z 1026.002,A -85,B 0,C 180,E1 -3499.196,E2 -3499.196} C_VEL
LIN {X 0,Y 671.994,Z 1032.962,A -85,B 0,C 180,E1 -3501.012,E2 -3501.012} C_VEL
LIN {X 0,Y 671.954,Z 1039.13,A -85,B 0,C 180,E1 -3502.991,E2 -3502.991} C_VEL
LIN {X 0,Y 671.914,Z 1043.732,A -85,B 0,C 180,E1 -3505.049,E2 -3505.049} C_VEL
LIN {X 0,Y 671.911,Z 1046.593,A -85,B 0,C 180,E1 -3506.904,E2 -3506.904} C_VEL
LIN {X 0,Y 671.909,Z 1048.249,A -85,B 0,C 180,E1 -3509.062,E2 -3509.062} C_VEL
LIN {X 0,Y 671.904,Z 1048.296,A -85,B 0,C 180,E1 -3510.853,E2 -3510.853} C_VEL
LIN {X 0,Y 671.906,Z 1046.97,A -85,B 0,C 180,E1 -3512.9,E2 -3512.9} C_VEL
LIN {X 0,Y 671.915,Z 1044.057,A -85,B 0,C 180,E1 -3514.866,E2 -3514.866} C_VEL
LIN {X 0,Y 671.928,Z 1040.178,A -85,B 0,C 180,E1 -3516.665,E2 -3516.665} C_VEL
LIN {X 0,Y 671.982,Z 1033.667,A -85,B 0,C 180,E1 -3518.878,E2 -3518.878} C_VEL
LIN {X 0,Y 672.094,Z 1027.081,A -85,B 0,C 180,E1 -3520.631,E2 -3520.631} C_VEL
LIN {X 0,Y 672.281,Z 1017.923,A -85,B 0,C 180,E1 -3522.662,E2 -3522.662} C_VEL
LIN {X 0,Y 672.538,Z 1007.523,A -85,B 0,C 180,E1 -3524.563,E2 -3524.563} C_VEL
LIN {X 0,Y 672.916,Z 995.362,A -85,B 0,C 180,E1 -3526.488,E2 -3526.488} C_VEL
LIN {X 0,Y 673.411,Z 981.579,A -85,B 0,C 180,E1 -3528.348,E2 -3528.348} C_VEL
LIN {X 0,Y 674.051,Z 966.578,A -85,B 0,C 180,E1 -3530.13,E2 -3530.13} C_VEL
LIN {X 0,Y 674.783,Z 949.988,A -85,B 0,C 180,E1 -3531.835,E2 -3531.835} C_VEL
LIN {X 0,Y 675.674,Z 932.147,A -85,B 0,C 180,E1 -3533.458,E2 -3533.458} C_VEL
LIN {X 0,Y 676.569,Z 913.81,A -85,B 0,C 180,E1 -3534.91,E2 -3534.91} C_VEL
LIN {X 0,Y 677.65,Z 893.605,A -85,B 0,C 180,E1 -3536.321,E2 -3536.321} C_VEL
LIN {X 0,Y 678.612,Z 874.091,A -85,B 0,C 180,E1 -3537.5,E2 -3537.5} C_VEL
LIN {X 0,Y 679.655,Z 853.096,A -85,B 0,C 180,E1 -3538.611,E2 -3538.611} C_VEL
LIN {X 0,Y 680.671,Z 830.395,A -85,B 0,C 180,E1 -3539.624,E2 -3539.624} C_VEL
LIN {X 0,Y 681.48,Z 811.392,A -85,B 0,C 180,E1 -3540.348,E2 -3540.348} C_VEL
LIN {X 0,Y 682.356,Z 786.362,A -85,B 0,C 180,E1 -3541.137,E2 -3541.137} C_VEL
LIN {X 0,Y 683.038,Z 764.657,A -85,B 0,C 180,E1 -3541.67,E2 -3541.67} C_VEL
LIN {X 0,Y 683.681,Z 739.731,A -85,B 0,C 180,E1 -3542.131,E2 -3542.131} C_VEL
LIN {X 0,Y 684.25,Z 683.6,A -85,B 0,C 180,E1 -3542.817,E2 -3542.817} C_VEL
LIN {X 0,Y 686.534,Z 434.555,A -85,B 0,C 180,E1 -3545.782,E2 -3545.782} C_VEL
LIN {X 0,Y 686.984,Z 367.151,A -85,B 0,C 180,E1 -3546.611,E2 -3546.611} C_VEL
LIN {X 0,Y 684.905,Z 362.773,A -85,B 0,C 180,E1 -3546.797,E2 -3546.797} C_VEL
LIN {X 0,Y 676.349,Z 347.946,A -85,B 0,C 180,E1 -3547.554,E2 -3547.554} C_VEL
LIN {X 0,Y 672.527,Z 337.46,A -85,B 0,C 180,E1 -3548.75,E2 -3548.75} C_VEL
LIN {X 0,Y 672.576,Z 337.454,A -85,B 0,C 180,E1 -3551.761,E2 -3551.761} C_VEL
LIN {X 0,Y 672.517,Z 337.44,A -85,B 0,C 180,E1 -3554.588,E2 -3554.588} C_VEL
LIN {X 0,Y 672.581,Z 337.44,A -85,B 0,C 180,E1 -3557.435,E2 -3557.435} C_VEL
LIN {X 0,Y 672.526,Z 337.451,A -85,B 0,C 180,E1 -3560.37,E2 -3560.37} C_VEL
LIN {X 0,Y 672.533,Z 337.451,A -85,B 0,C 180,E1 -3563.083,E2 -3563.083} C_VEL
LIN {X 0,Y 672.547,Z 337.45,A -85,B 0,C 180,E1 -3566.218,E2 -3566.218} C_VEL
LIN {X 0,Y 672.52,Z 337.45,A -85,B 0,C 180,E1 -3568.941,E2 -3568.941} C_VEL
LIN {X 0,Y 672.59,Z 337.444,A -85,B 0,C 180,E1 -3571.884,E2 -3571.884} C_VEL
LIN {X 0,Y 672.519,Z 337.453,A -85,B 0,C 180,E1 -3574.741,E2 -3574.741} C_VEL
LIN {X 0,Y 672.544,Z 337.451,A -85,B 0,C 180,E1 -3577.445,E2 -3577.445} C_VEL
LIN {X 0,Y 672.538,Z 337.445,A -85,B 0,C 180,E1 -3580.547,E2 -3580.547} C_VEL
LIN {X 0,Y 672.521,Z 337.454,A -85,B 0,C 180,E1 -3583.236,E2 -3583.236} C_VEL
LIN {X 0,Y 672.585,Z 337.45,A -85,B 0,C 180,E1 -3586.24,E2 -3586.24} C_VEL
LIN {X 0,Y 672.516,Z 337.445,A -85,B 0,C 180,E1 -3589.116,E2 -3589.116} C_VEL
LIN {X 0,Y 672.578,Z 337.454,A -85,B 0,C 180,E1 -3591.967,E2 -3591.967} C_VEL
LIN {X 0,Y 672.524,Z 337.45,A -85,B 0,C 180,E1 -3594.968,E2 -3594.968} C_VEL
LIN {X 0,Y 672.536,Z 337.453,A -85,B 0,C 180,E1 -3597.699,E2 -3597.699} C_VEL
LIN {X 0,Y 672.542,Z 337.451,A -85,B 0,C 180,E1 -3600.852,E2 -3600.852} C_VEL
LIN {X 0,Y 672.52,Z 337.444,A -85,B 0,C 180,E1 -3603.58,E2 -3603.58} C_VEL
LIN {X 0,Y 672.59,Z 337.444,A -85,B 0,C 180,E1 -3606.573,E2 -3606.573} C_VEL
LIN {X 0,Y 672.517,Z 337.452,A -85,B 0,C 180,E1 -3609.413,E2 -3609.413} C_VEL
LIN {X 0,Y 672.572,Z 337.447,A -85,B 0,C 180,E1 -3612.274,E2 -3612.274} C_VEL
LIN {X 0,Y 672.526,Z 337.45,A -85,B 0,C 180,E1 -3615.258,E2 -3615.258} C_VEL
LIN {X 0,Y 672.524,Z 337.451,A -85,B 0,C 180,E1 -3617.925,E2 -3617.925} C_VEL
LIN {X 0,Y 672.563,Z 337.447,A -85,B 0,C 180,E1 -3620.995,E2 -3620.995} C_VEL
LIN {X 0,Y 672.516,Z 337.451,A -85,B 0,C 180,E1 -3623.761,E2 -3623.761} C_VEL
LIN {X 0,Y 672.588,Z 337.451,A -85,B 0,C 180,E1 -3626.688,E2 -3626.688} C_VEL
LIN {X 0,Y 672.522,Z 337.453,A -85,B 0,C 180,E1 -3629.578,E2 -3629.578} C_VEL
LIN {X 0,Y 672.532,Z 337.452,A -85,B 0,C 180,E1 -3632.259,E2 -3632.259} C_VEL
LIN {X 0,Y 672.539,Z 337.453,A -85,B 0,C 180,E1 -3635.439,E2 -3635.439} C_VEL
LIN {X 0,Y 672.52,Z 337.454,A -85,B 0,C 180,E1 -3638.14,E2 -3638.14} C_VEL
LIN {X 0,Y 672.587,Z 337.432,A -85,B 0,C 180,E1 -3641.086,E2 -3641.086} C_VEL
LIN {X 0,Y 672.517,Z 337.452,A -85,B 0,C 180,E1 -3643.978,E2 -3643.978} C_VEL
LIN {X 0,Y 672.561,Z 337.455,A -85,B 0,C 180,E1 -3646.759,E2 -3646.759} C_VEL
LIN {X 0,Y 672.593,Z 337.469,A -85,B 0,C 180,E1 -3649.174,E2 -3649.174} C_VEL
LIN {X 0,Y 682.604,Z 364.169,A -85,B 0,C 180,E1 -3651.955,E2 -3651.955} C_VEL
LIN {X 0,Y 682.307,Z 376.94,A -85,B 0,C 180,E1 -3652.891,E2 -3652.891} C_VEL
LIN {X 0,Y 687.168,Z 397.583,A -85,B 0,C 180,E1 -3653.458,E2 -3653.458} C_VEL
LIN {X 0,Y 684.718,Z 660.042,A -85,B 0,C 180,E1 -3656.596,E2 -3656.596} C_VEL
LIN {X 0,Y 683.699,Z 767.706,A -85,B 0,C 180,E1 -3657.886,E2 -3657.886} C_VEL
LIN {X 0,Y 683.091,Z 793.143,A -85,B 0,C 180,E1 -3658.342,E2 -3658.342} C_VEL
LIN {X 0,Y 682.413,Z 814.553,A -85,B 0,C 180,E1 -3658.86,E2 -3658.86} C_VEL
LIN {X 0,Y 681.586,Z 838.967,A -85,B 0,C 180,E1 -3659.61,E2 -3659.61} C_VEL
LIN {X 0,Y 680.717,Z 859.346,A -85,B 0,C 180,E1 -3660.378,E2 -3660.378} C_VEL
LIN {X 0,Y 679.795,Z 880.264,A -85,B 0,C 180,E1 -3661.299,E2 -3661.299} C_VEL
LIN {X 0,Y 678.692,Z 902.316,A -85,B 0,C 180,E1 -3662.445,E2 -3662.445} C_VEL
LIN {X 0,Y 677.757,Z 921.216,A -85,B 0,C 180,E1 -3663.574,E2 -3663.574} C_VEL
LIN {X 0,Y 676.663,Z 942.008,A -85,B 0,C 180,E1 -3665,E2 -3665} C_VEL
LIN {X 0,Y 675.801,Z 959.399,A -85,B 0,C 180,E1 -3666.362,E2 -3666.362} C_VEL
LIN {X 0,Y 674.844,Z 978.605,A -85,B 0,C 180,E1 -3668.076,E2 -3668.076} C_VEL
LIN {X 0,Y 674.17,Z 993.722,A -85,B 0,C 180,E1 -3669.611,E2 -3669.611} C_VEL
LIN {X 0,Y 673.468,Z 1009.816,A -85,B 0,C 180,E1 -3671.475,E2 -3671.475} C_VEL
LIN {X 0,Y 673.008,Z 1022.525,A -85,B 0,C 180,E1 -3673.159,E2 -3673.159} C_VEL
LIN {X 0,Y 672.583,Z 1035.763,A -85,B 0,C 180,E1 -3675.185,E2 -3675.185} C_VEL
LIN {X 0,Y 672.325,Z 1045.586,A -85,B 0,C 180,E1 -3676.939,E2 -3676.939} C_VEL
LIN {X 0,Y 672.115,Z 1055.476,A -85,B 0,C 180,E1 -3679.022,E2 -3679.022} C_VEL
LIN {X 0,Y 672.011,Z 1062.514,A -85,B 0,C 180,E1 -3680.839,E2 -3680.839} C_VEL
LIN {X 0,Y 671.957,Z 1068.761,A -85,B 0,C 180,E1 -3682.82,E2 -3682.82} C_VEL
LIN {X 0,Y 671.924,Z 1073.497,A -85,B 0,C 180,E1 -3684.877,E2 -3684.877} C_VEL
LIN {X 0,Y 671.916,Z 1076.462,A -85,B 0,C 180,E1 -3686.758,E2 -3686.758} C_VEL
LIN {X 0,Y 671.914,Z 1078.238,A -85,B 0,C 180,E1 -3688.977,E2 -3688.977} C_VEL
LIN {X 0,Y 671.899,Z 1078.306,A -85,B 0,C 180,E1 -3690.767,E2 -3690.767} C_VEL
LIN {X 0,Y 671.909,Z 1077.017,A -85,B 0,C 180,E1 -3692.815,E2 -3692.815} C_VEL
LIN {X 0,Y 671.922,Z 1073.974,A -85,B 0,C 180,E1 -3694.866,E2 -3694.866} C_VEL
LIN {X 0,Y 671.923,Z 1070.07,A -85,B 0,C 180,E1 -3696.665,E2 -3696.665} C_VEL
LIN {X 0,Y 671.979,Z 1063.726,A -85,B 0,C 180,E1 -3698.816,E2 -3698.816} C_VEL
LIN {X 0,Y 672.097,Z 1056.896,A -85,B 0,C 180,E1 -3700.631,E2 -3700.631} C_VEL
LIN {X 0,Y 672.282,Z 1047.687,A -85,B 0,C 180,E1 -3702.662,E2 -3702.662} C_VEL
LIN {X 0,Y 672.539,Z 1037.261,A -85,B 0,C 180,E1 -3704.563,E2 -3704.563} C_VEL
LIN {X 0,Y 672.919,Z 1025.064,A -85,B 0,C 180,E1 -3706.487,E2 -3706.487} C_VEL
LIN {X 0,Y 673.424,Z 1011.228,A -85,B 0,C 180,E1 -3708.347,E2 -3708.347} C_VEL
LIN {X 0,Y 674.071,Z 996.17,A -85,B 0,C 180,E1 -3710.129,E2 -3710.129} C_VEL
LIN {X 0,Y 674.759,Z 980.46,A -85,B 0,C 180,E1 -3711.744,E2 -3711.744} C_VEL
LIN {X 0,Y 675.65,Z 962.716,A -85,B 0,C 180,E1 -3713.366,E2 -3713.366} C_VEL
LIN {X 0,Y 676.557,Z 944.068,A -85,B 0,C 180,E1 -3714.846,E2 -3714.846} C_VEL
LIN {X 0,Y 677.598,Z 924.669,A -85,B 0,C 180,E1 -3716.208,E2 -3716.208} C_VEL
LIN {X 0,Y 678.618,Z 903.937,A -85,B 0,C 180,E1 -3717.463,E2 -3717.463} C_VEL
LIN {X 0,Y 679.68,Z 882.638,A -85,B 0,C 180,E1 -3718.59,E2 -3718.59} C_VEL
LIN {X 0,Y 680.68,Z 860.266,A -85,B 0,C 180,E1 -3719.585,E2 -3719.585} C_VEL
LIN {X 0,Y 681.546,Z 839.836,A -85,B 0,C 180,E1 -3720.359,E2 -3720.359} C_VEL
LIN {X 0,Y 682.405,Z 814.779,A -85,B 0,C 180,E1 -3721.134,E2 -3721.134} C_VEL
LIN {X 0,Y 683.085,Z 793.284,A -85,B 0,C 180,E1 -3721.656,E2 -3721.656} C_VEL
LIN {X 0,Y 683.699,Z 767.826,A -85,B 0,C 180,E1 -3722.113,E2 -3722.113} C_VEL
LIN {X 0,Y 684.654,Z 667.5,A -85,B 0,C 180,E1 -3723.315,E2 -3723.315} C_VEL
LIN {X 0,Y 687.132,Z 401.373,A -85,B 0,C 180,E1 -3726.497,E2 -3726.497} C_VEL
LIN {X 0,Y 686.935,Z 395.796,A -85,B 0,C 180,E1 -3726.58,E2 -3726.58} C_VEL
LIN {X 0,Y 682.241,Z 376.223,A -85,B 0,C 180,E1 -3727.144,E2 -3727.144} C_VEL
LIN {X 0,Y 682.47,Z 363.78,A -85,B 0,C 180,E1 -3728.083,E2 -3728.083} C_VEL
LIN {X 0,Y 674.92,Z 343.937,A -85,B 0,C 180,E1 -3730.141,E2 -3730.141} C_VEL
LIN {X 0,Y 672.59,Z 337.449,A -85,B 0,C 180,E1 -3730.852,E2 -3730.852} C_VEL
LIN {X 0,Y 672.52,Z 337.455,A -85,B 0,C 180,E1 -3733.737,E2 -3733.737} C_VEL
LIN {X 0,Y 672.536,Z 337.453,A -85,B 0,C 180,E1 -3736.389,E2 -3736.389} C_VEL
LIN {X 0,Y 672.535,Z 337.453,A -85,B 0,C 180,E1 -3739.592,E2 -3739.592} C_VEL
LIN {X 0,Y 672.522,Z 337.452,A -85,B 0,C 180,E1 -3742.276,E2 -3742.276} C_VEL
LIN {X 0,Y 672.578,Z 337.43,A -85,B 0,C 180,E1 -3745.297,E2 -3745.297} C_VEL
LIN {X 0,Y 672.517,Z 337.449,A -85,B 0,C 180,E1 -3748.142,E2 -3748.142} C_VEL
LIN {X 0,Y 672.573,Z 337.449,A -85,B 0,C 180,E1 -3750.945,E2 -3750.945} C_VEL
LIN {X 0,Y 672.528,Z 337.454,A -85,B 0,C 180,E1 -3753.986,E2 -3753.986} C_VEL
LIN {X 0,Y 672.535,Z 337.447,A -85,B 0,C 180,E1 -3756.704,E2 -3756.704} C_VEL
LIN {X 0,Y 672.539,Z 337.451,A -85,B 0,C 180,E1 -3759.913,E2 -3759.913} C_VEL
LIN {X 0,Y 672.526,Z 337.451,A -85,B 0,C 180,E1 -3762.65,E2 -3762.65} C_VEL
LIN {X 0,Y 672.578,Z 337.456,A -85,B 0,C 180,E1 -3765.713,E2 -3765.713} C_VEL
LIN {X 0,Y 672.519,Z 337.447,A -85,B 0,C 180,E1 -3768.508,E2 -3768.508} C_VEL
LIN {X 0,Y 672.584,Z 337.449,A -85,B 0,C 180,E1 -3771.364,E2 -3771.364} C_VEL
LIN {X 0,Y 672.526,Z 337.454,A -85,B 0,C 180,E1 -3774.369,E2 -3774.369} C_VEL
LIN {X 0,Y 672.541,Z 337.445,A -85,B 0,C 180,E1 -3777.103,E2 -3777.103} C_VEL
LIN {X 0,Y 672.542,Z 337.453,A -85,B 0,C 180,E1 -3780.256,E2 -3780.256} C_VEL
LIN {X 0,Y 672.526,Z 337.447,A -85,B 0,C 180,E1 -3782.983,E2 -3782.983} C_VEL
LIN {X 0,Y 672.585,Z 337.447,A -85,B 0,C 180,E1 -3785.98,E2 -3785.98} C_VEL
LIN {X 0,Y 672.522,Z 337.453,A -85,B 0,C 180,E1 -3788.809,E2 -3788.809} C_VEL
LIN {X 0,Y 672.576,Z 337.442,A -85,B 0,C 180,E1 -3791.665,E2 -3791.665} C_VEL
LIN {X 0,Y 672.527,Z 337.45,A -85,B 0,C 180,E1 -3794.728,E2 -3794.728} C_VEL
LIN {X 0,Y 672.546,Z 337.449,A -85,B 0,C 180,E1 -3797.477,E2 -3797.477} C_VEL
LIN {X 0,Y 672.543,Z 337.454,A -85,B 0,C 180,E1 -3800.632,E2 -3800.632} C_VEL
LIN {X 0,Y 672.532,Z 337.448,A -85,B 0,C 180,E1 -3803.389,E2 -3803.389} C_VEL
LIN {X 0,Y 672.569,Z 337.453,A -85,B 0,C 180,E1 -3806.495,E2 -3806.495} C_VEL
LIN {X 0,Y 672.526,Z 337.452,A -85,B 0,C 180,E1 -3809.285,E2 -3809.285} C_VEL
LIN {X 0,Y 672.589,Z 337.445,A -85,B 0,C 180,E1 -3812.233,E2 -3812.233} C_VEL
LIN {X 0,Y 672.526,Z 337.452,A -85,B 0,C 180,E1 -3813.403,E2 -3813.403} C_VEL
LIN {X 0,Y 671.559,Z 337.577,A -85,B 0,C 180,E1 -3814.059,E2 -3814.059} C_VEL
LIN {X 0,Y 665.183,Z 338.369,A -85,B 0,C 180,E1 -3815.898,E2 -3815.898} C_VEL
LIN {X 0,Y 664.65,Z 338.441,A -85,B 0,C 180,E1 -3816.376,E2 -3816.376} C_VEL
LIN {X 0,Y 664.587,Z 338.442,A -85,B 0,C 180,E1 -3819.347,E2 -3819.347} C_VEL
LIN {X 0,Y 664.648,Z 338.44,A -85,B 0,C 180,E1 -3822.258,E2 -3822.258} C_VEL
LIN {X 0,Y 664.592,Z 338.443,A -85,B 0,C 180,E1 -3825.246,E2 -3825.246} C_VEL
LIN {X 0,Y 664.611,Z 338.443,A -85,B 0,C 180,E1 -3828.006,E2 -3828.006} C_VEL
LIN {X 0,Y 664.637,Z 338.457,A -85,B 0,C 180,E1 -3830.884,E2 -3830.884} C_VEL
LIN {X 0,Y 668.49,Z 348.838,A -85,B 0,C 180,E1 -3832.041,E2 -3832.041} C_VEL
LIN {X 0,Y 680.725,Z 370.023,A -85,B 0,C 180,E1 -3833.122,E2 -3833.122} C_VEL
LIN {X 0,Y 678.233,Z 610.68,A -85,B 0,C 180,E1 -3836.038,E2 -3836.038} C_VEL
LIN {X 0,Y 676.919,Z 737.536,A -85,B 0,C 180,E1 -3837.567,E2 -3837.567} C_VEL
LIN {X 0,Y 676.264,Z 762.968,A -85,B 0,C 180,E1 -3838.025,E2 -3838.025} C_VEL
LIN {X 0,Y 675.54,Z 784.182,A -85,B 0,C 180,E1 -3838.541,E2 -3838.541} C_VEL
LIN {X 0,Y 674.642,Z 808.071,A -85,B 0,C 180,E1 -3839.275,E2 -3839.275} C_VEL
LIN {X 0,Y 673.7,Z 828.311,A -85,B 0,C 180,E1 -3840.038,E2 -3840.038} C_VEL
LIN {X 0,Y 672.742,Z 848.357,A -85,B 0,C 180,E1 -3840.921,E2 -3840.921} C_VEL
LIN {X 0,Y 671.469,Z 871.554,A -85,B 0,C 180,E1 -3842.123,E2 -3842.123} C_VEL
LIN {X 0,Y 670.407,Z 891.162,A -85,B 0,C 180,E1 -3843.303,E2 -3843.303} C_VEL
LIN {X 0,Y 669.165,Z 912.642,A -85,B 0,C 180,E1 -3844.795,E2 -3844.795} C_VEL
LIN {X 0,Y 668.215,Z 929.977,A -85,B 0,C 180,E1 -3846.171,E2 -3846.171} C_VEL
LIN {X 0,Y 667.201,Z 948.483,A -85,B 0,C 180,E1 -3847.844,E2 -3847.844} C_VEL
LIN {X 0,Y 666.412,Z 964.064,A -85,B 0,C 180,E1 -3849.446,E2 -3849.446} C_VEL
LIN {X 0,Y 665.637,Z 980.176,A -85,B 0,C 180,E1 -3851.34,E2 -3851.34} C_VEL
LIN {X 0,Y 665.112,Z 993.478,A -85,B 0,C 180,E1 -3853.133,E2 -3853.133} C_VEL
LIN {X 0,Y 664.646,Z 1006.546,A -85,B 0,C 180,E1 -3855.182,E2 -3855.182} C_VEL
LIN {X 0,Y 664.353,Z 1016.251,A -85,B 0,C 180,E1 -3856.953,E2 -3856.953} C_VEL
LIN {X 0,Y 664.123,Z 1026.005,A -85,B 0,C 180,E1 -3859.065,E2 -3859.065} C_VEL
LIN {X 0,Y 664.013,Z 1032.964,A -85,B 0,C 180,E1 -3860.903,E2 -3860.903} C_VEL
LIN {X 0,Y 663.957,Z 1039.344,A -85,B 0,C 180,E1 -3862.994,E2 -3862.994} C_VEL
LIN {X 0,Y 663.917,Z 1043.732,A -85,B 0,C 180,E1 -3864.989,E2 -3864.989} C_VEL
LIN {X 0,Y 663.91,Z 1046.516,A -85,B 0,C 180,E1 -3866.806,E2 -3866.806} C_VEL
LIN {X 0,Y 663.913,Z 1048.226,A -85,B 0,C 180,E1 -3868.965,E2 -3868.965} C_VEL
LIN {X 0,Y 663.899,Z 1048.318,A -85,B 0,C 180,E1 -3870.777,E2 -3870.777} C_VEL
LIN {X 0,Y 663.899,Z 1047.126,A -85,B 0,C 180,E1 -3872.763,E2 -3872.763} C_VEL
LIN {X 0,Y 663.917,Z 1044.215,A -85,B 0,C 180,E1 -3874.838,E2 -3874.838} C_VEL
LIN {X 0,Y 663.93,Z 1040.384,A -85,B 0,C 180,E1 -3876.659,E2 -3876.659} C_VEL
LIN {X 0,Y 663.984,Z 1034.488,A -85,B 0,C 180,E1 -3878.748,E2 -3878.748} C_VEL
LIN {X 0,Y 664.11,Z 1027.433,A -85,B 0,C 180,E1 -3880.672,E2 -3880.672} C_VEL
LIN {X 0,Y 664.3,Z 1018.918,A -85,B 0,C 180,E1 -3882.606,E2 -3882.606} C_VEL
LIN {X 0,Y 664.605,Z 1007.912,A -85,B 0,C 180,E1 -3884.672,E2 -3884.672} C_VEL
LIN {X 0,Y 664.989,Z 996.519,A -85,B 0,C 180,E1 -3886.51,E2 -3886.51} C_VEL
LIN {X 0,Y 665.559,Z 982.273,A -85,B 0,C 180,E1 -3888.481,E2 -3888.481} C_VEL
LIN {X 0,Y 666.216,Z 968.133,A -85,B 0,C 180,E1 -3890.194,E2 -3890.194} C_VEL
LIN {X 0,Y 667.025,Z 951.833,A -85,B 0,C 180,E1 -3891.917,E2 -3891.917} C_VEL
LIN {X 0,Y 667.871,Z 935.983,A -85,B 0,C 180,E1 -3893.401,E2 -3893.401} C_VEL
LIN {X 0,Y 668.969,Z 916.234,A -85,B 0,C 180,E1 -3895.024,E2 -3895.024} C_VEL
LIN {X 0,Y 670.03,Z 897.701,A -85,B 0,C 180,E1 -3896.357,E2 -3896.357} C_VEL
LIN {X 0,Y 671.232,Z 876.317,A -85,B 0,C 180,E1 -3897.695,E2 -3897.695} C_VEL
LIN {X 0,Y 672.276,Z 856.683,A -85,B 0,C 180,E1 -3898.76,E2 -3898.76} C_VEL
LIN {X 0,Y 673.492,Z 833.011,A -85,B 0,C 180,E1 -3899.858,E2 -3899.858} C_VEL
LIN {X 0,Y 674.39,Z 813.57,A -85,B 0,C 180,E1 -3900.617,E2 -3900.617} C_VEL
LIN {X 0,Y 675.335,Z 791.007,A -85,B 0,C 180,E1 -3901.361,E2 -3901.361} C_VEL
LIN {X 0,Y 676.114,Z 766.975,A -85,B 0,C 180,E1 -3901.977,E2 -3901.977} C_VEL
LIN {X 0,Y 676.793,Z 744.122,A -85,B 0,C 180,E1 -3902.422,E2 -3902.422} C_VEL
LIN {X 0,Y 677.271,Z 709.975,A -85,B 0,C 180,E1 -3902.871,E2 -3902.871} C_VEL
LIN {X 0,Y 679.843,Z 454.709,A -85,B 0,C 180,E1 -3905.933,E2 -3905.933} C_VEL
LIN {X 0,Y 680.605,Z 369.663,A -85,B 0,C 180,E1 -3906.981,E2 -3906.981} C_VEL
LIN {X 0,Y 668.235,Z 348.247,A -85,B 0,C 180,E1 -3908.088,E2 -3908.088} C_VEL
LIN {X 0,Y 664.637,Z 338.438,A -85,B 0,C 180,E1 -3909.215,E2 -3909.215} C_VEL
LIN {X 0,Y 664.587,Z 338.446,A -85,B 0,C 180,E1 -3912.262,E2 -3912.262} C_VEL
LIN {X 0,Y 664.598,Z 338.43,A -85,B 0,C 180,E1 -3915.001,E2 -3915.001} C_VEL
LIN {X 0,Y 664.596,Z 338.421,A -85,B 0,C 180,E1 -3918.202,E2 -3918.202} C_VEL
LIN {X 0,Y 664.586,Z 338.443,A -85,B 0,C 180,E1 -3920.927,E2 -3920.927} C_VEL
LIN {X 0,Y 664.626,Z 338.44,A -85,B 0,C 180,E1 -3924.036,E2 -3924.036} C_VEL
LIN {X 0,Y 664.579,Z 338.441,A -85,B 0,C 180,E1 -3926.794,E2 -3926.794} C_VEL
LIN {X 0,Y 664.653,Z 338.438,A -85,B 0,C 180,E1 -3929.737,E2 -3929.737} C_VEL
LIN {X 0,Y 664.582,Z 338.434,A -85,B 0,C 180,E1 -3932.685,E2 -3932.685} C_VEL
LIN {X 0,Y 664.601,Z 338.445,A -85,B 0,C 180,E1 -3935.371,E2 -3935.371} C_VEL
LIN {X 0,Y 664.596,Z 338.44,A -85,B 0,C 180,E1 -3938.556,E2 -3938.556} C_VEL
LIN {X 0,Y 664.583,Z 338.437,A -85,B 0,C 180,E1 -3941.218,E2 -3941.218} C_VEL
LIN {X 0,Y 664.646,Z 338.43,A -85,B 0,C 180,E1 -3944.199,E2 -3944.199} C_VEL
LIN {X 0,Y 664.579,Z 338.442,A -85,B 0,C 180,E1 -3947.045,E2 -3947.045} C_VEL
LIN {X 0,Y 664.639,Z 338.435,A -85,B 0,C 180,E1 -3949.95,E2 -3949.95} C_VEL
LIN {X 0,Y 664.586,Z 338.436,A -85,B 0,C 180,E1 -3952.913,E2 -3952.913} C_VEL
LIN {X 0,Y 664.591,Z 338.442,A -85,B 0,C 180,E1 -3955.599,E2 -3955.599} C_VEL
LIN {X 0,Y 664.615,Z 338.434,A -85,B 0,C 180,E1 -3958.707,E2 -3958.707} C_VEL
LIN {X 0,Y 664.579,Z 338.443,A -85,B 0,C 180,E1 -3961.466,E2 -3961.466} C_VEL
LIN {X 0,Y 664.647,Z 338.44,A -85,B 0,C 180,E1 -3964.487,E2 -3964.487} C_VEL
LIN {X 0,Y 664.577,Z 338.436,A -85,B 0,C 180,E1 -3967.348,E2 -3967.348} C_VEL
LIN {X 0,Y 664.621,Z 338.444,A -85,B 0,C 180,E1 -3970.138,E2 -3970.138} C_VEL
LIN {X 0,Y 664.587,Z 338.438,A -85,B 0,C 180,E1 -3973.237,E2 -3973.237} C_VEL
LIN {X 0,Y 664.588,Z 338.442,A -85,B 0,C 180,E1 -3975.892,E2 -3975.892} C_VEL
LIN {X 0,Y 664.623,Z 338.437,A -85,B 0,C 180,E1 -3978.963,E2 -3978.963} C_VEL
LIN {X 0,Y 664.579,Z 338.439,A -85,B 0,C 180,E1 -3981.723,E2 -3981.723} C_VEL
LIN {X 0,Y 664.648,Z 338.435,A -85,B 0,C 180,E1 -3984.628,E2 -3984.628} C_VEL
LIN {X 0,Y 664.581,Z 338.438,A -85,B 0,C 180,E1 -3987.607,E2 -3987.607} C_VEL
LIN {X 0,Y 664.6,Z 338.445,A -85,B 0,C 180,E1 -3990.279,E2 -3990.279} C_VEL
LIN {X 0,Y 664.601,Z 338.44,A -85,B 0,C 180,E1 -3993.412,E2 -3993.412} C_VEL
LIN {X 0,Y 664.582,Z 338.445,A -85,B 0,C 180,E1 -3996.142,E2 -3996.142} C_VEL
LIN {X 0,Y 664.639,Z 338.433,A -85,B 0,C 180,E1 -3999.187,E2 -3999.187} C_VEL
LIN {X 0,Y 664.577,Z 338.438,A -85,B 0,C 180,E1 -4002.031,E2 -4002.031} C_VEL
LIN {X 0,Y 664.641,Z 338.442,A -85,B 0,C 180,E1 -4004.881,E2 -4004.881} C_VEL
LIN {X 0,Y 664.583,Z 338.443,A -85,B 0,C 180,E1 -4007.88,E2 -4007.88} C_VEL
LIN {X 0,Y 664.614,Z 338.491,A -85,B 0,C 180,E1 -4008.683,E2 -4008.683} C_VEL
LIN {X 0,Y 673.669,Z 362.524,A -85,B 0,C 180,E1 -4011.251,E2 -4011.251} C_VEL
LIN {X 0,Y 675.568,Z 368.029,A -85,B 0,C 180,E1 -4011.806,E2 -4011.806} C_VEL
LIN {X 0,Y 675.405,Z 376.849,A -85,B 0,C 180,E1 -4012.448,E2 -4012.448} C_VEL
LIN {X 0,Y 680.703,Z 399.359,A -85,B 0,C 180,E1 -4013.079,E2 -4013.079} C_VEL
LIN {X 0,Y 678.007,Z 663.213,A -85,B 0,C 180,E1 -4016.261,E2 -4016.261} C_VEL
LIN {X 0,Y 676.914,Z 767.813,A -85,B 0,C 180,E1 -4017.526,E2 -4017.526} C_VEL
